screen "1.4.2_DR3_Advanced_Scale_Parameters_2" 800x480, template "Template_1"
   TextField "OBJECT_33" at 0,0 size 595x34; Text '1.4.2 Erweiterte Waagenparameter 2 von 5 / 1.4.2 Advanced Scale Parameter 2 of 5 / 1.4.2 Tous les paramètres 2/5 / Setup 1/3'
   Button "Exit_to_service_1" at 670,390 size 80x80; TextOn 'Texte / text'; TextOff 'Texte / text'; PictureOff "Right"
      on Press: ActivateScreen("1.4.3_DR3_Advanced_Scale_Parameters_3", 0)
   Button "Exit_to_service_2" at 545,390 size 80x80; TextOn 'Texte / text'; TextOff 'Texte / text'; PictureOff "Left"
      on Press: ActivateScreen("1.4.1_DR3_Advanced_Scale_Parameters_1", 0)
   Group "Group" at 700,5 size 95x30; Text 'Service'; PictureList "Signal_grey_yellow"
   Button "Exit_to_service" at 45,390 size 80x80; TextOn 'Texte / text'; TextOff 'Texte / text'; PictureOff "Exit"
      on Release: ActivateScreen("1.0_Menu_setup", 0)
      on Press: SetTag("WP231PR_DB_s_CMD2_i_CMD_CODE", '2'); SetBit("WP231PR_DB_s_CMD2_bo_CMD_TRIGGER")
   Button "OBJECT_13" at 360,390 size 80x80; TextOn 'Texte / text'; TextOff 'Texte / text'; PictureOff "Save"
      on Press: SetTag("WP231PR_DB_s_CMD2_i_CMD_CODE", '4003'); SetBit("WP231PR_DB_s_CMD2_bo_CMD_TRIGGER")
   TextField "OBJECT_306" at 172,114 size 279x26; Text 'Einschaltnullsetzen / Initial Zeroing / RAZ initiale / Scale name'
   TextField "OBJECT_7" at 69,155 size 380x26; Text 'Einschaltnullsetzen bei tarierter Waage / Initial zeroing if scale is tared / RAZ initiale quand la balance est tarée / Weight Unit'
   SymbolicIOField "Symbolisches EA-Feld_1" at 464,110 size 110x31; TextOn '1'; HelpText 'Die Waage kann durch einen Neustart automatisch nullgestellt werden. / The scale can be zeroed automatically by a power on. / La balance peut être remise à zéro à la mise sous tension'; TextOff '0'; TextList "003072_NO_YES"
      ProcessValue <- "WP231PR_DB_DR03_INITIAL_ZEROING"
   SymbolicIOField "Symbolisches EA-Feld_2" at 464,151 size 110x31; TextOn '1'; HelpText 'Shall the scale be zeroed by power on if it was tared? / RAZ à la mise sous tension lorsque la tare >< 0?'; TextOff '0'; TextList "003072_NO_YES"
      ProcessValue <- "WP231PR_DB_DR03_INITIAL_ZEROING_IF_TARED"
   TextField "OBJECT_3" at 25,199 size 426x26; Text 'Negativer Nullsetzgrenzwert (Einschaltnullsetzen) / Negative zeroing limit (initital zeroing) / Limite négative de RAZ (RAZ initiale) / Weight Unit'
      Visibility <- "WP231PR_DB_DR03_INITIAL_ZEROING"
   TextField "OBJECT_6" at 52,242 size 399x26; Text 'Positiver Nullsetzgrenzwert (Einschaltnullsetzen) / Positive zeroing limit (initial zeroing) / Limite positive de RAZ (RAZ initiale) / Weight Unit'
      Visibility <- "WP231PR_DB_DR03_INITIAL_ZEROING"
   IOField "OBJECT_28" at 464,191 size 110x40; HelpText 'Negative Begrenzung des Nullstellwerts nach Einschalten der Waage. / Limite négative de la RAZ à la mise sous tension'; FormatPattern 99.99
      ProcessValue <- "WP231PR_DB_DR03_INITIAL_ZEROING_LIM_NEG"
      Visibility <- "WP231PR_DB_DR03_INITIAL_ZEROING"
   IOField "OBJECT_8" at 464,235 size 110x40; HelpText 'Positive Begrenzung des Nullstellwerts nach Einschalten der Waage. / Plage RAZ positive après mise sous tension'; FormatPattern 99.99
      ProcessValue <- "WP231PR_DB_DR03_INITIAL_ZEROING_LIM_POS"
      Visibility <- "WP231PR_DB_DR03_INITIAL_ZEROING"
   TextField "OBJECT_2" at 194,75 size 257x26; Text 'Automatische Nullnachführung / Automatic Zero Tracking / Maintien du zéro (zéro suiveur) / Weight Unit'
   SymbolicIOField "Symbolisches EA-Feld_3" at 464,71 size 110x31; TextOn '1'; HelpText 'Driftet die Waage weniger als 1/4d pro Sekunde stellt sie automatisch null. ACHTUNG: Bei langsamer Drift kann eine volle Waage mit 0kg angezeigt werden! If the scale drifts less than 1/4d per second, it'll be zeroed automatically. ATTENTION: A slow drift can effect, that the scale shows 0kg even if it's full! La balance effectue automatiquement une RAZ quand le poids dérive de moins de 1/4d par sec'; TextOff '0'; TextList "003072_NO_YES"
      ProcessValue <- "WP231PR_DB_DR03_ZERO_TRACKING"
   TextField "OBJECT_4" at 12,330 size 440x26; Text 'Positiver Nullstellgrenzwert (halbselbstt. Nullstellen) / Positive zeroing limit (semi-automatic zeroing) / Limite positive de RAZ (RAZ semi-automatique) / Scale name'
   TextField "OBJECT_9" at 13,287 size 439x26; Text 'Negativer Nullstellgrenzwert (halbselbstt. Nullstellen) / Negative zeroing limit (semi-automatic zeroing) / Limite négative de RAZ (RAZ semi-automatique) / Weight Unit'
   IOField "OBJECT_10" at 464,323 size 110x40; HelpText 'Positive Begrenzung des Nullstellwerts der Waage. / Plage RAZ positive'; FormatPattern 99.99
      ProcessValue <- "WP231PR_DB_DR03_SEM_AUT_ZERO_LIM_POS"
   IOField "OBJECT_11" at 464,279 size 110x40; HelpText 'Negative Begrenzung des Nullstellwerts der Waage. / Limite négative de la RAZ'; FormatPattern 99.99
      ProcessValue <- "WP231PR_DB_DR03_SEM_AUT_ZERO_LIM_NEG"
   TextField "OBJECT_22" at 575,199 size 22x26; Text '% / Calibration Weight'
      Visibility <- "WP231PR_DB_DR03_INITIAL_ZEROING"
   TextField "OBJECT_1" at 576,243 size 22x26; Text '% / Calibration Weight'
      Visibility <- "WP231PR_DB_DR03_INITIAL_ZEROING"
   TextField "OBJECT_5" at 578,286 size 22x26; Text '% / Calibration Weight'
   TextField "OBJECT_12" at 577,331 size 22x26; Text '% / Calibration Weight'
   Group "Group_3" at 599,286 size 166x26; Text 'von'
   Group "Group_4" at 599,329 size 166x26; Text 'von'
   IOField "OBJECT_15" at 631,245 size 85x23; FormatPattern 9999999.9
      Visibility <- "WP231PR_DB_DR03_INITIAL_ZEROING"
      ProcessValue <- "WP231PR_DB_DR03_MAX_WEIGHT"
   TextField "Textfeld_2" at 599,243 size 30x25; Text 'von / of / de'
      Visibility <- "WP231PR_DB_DR03_INITIAL_ZEROING"
   IOField "I/O field_1" at 699,244 size 66x25; FormatPattern ????
      Visibility <- "WP231PR_DB_DR03_INITIAL_ZEROING"
      ProcessValue <- "WP231PR_DB_DR03_WEIGHT_UNIT"
   IOField "OBJECT_14" at 631,202 size 85x23; FormatPattern 9999999.9
      Visibility <- "WP231PR_DB_DR03_INITIAL_ZEROING"
      ProcessValue <- "WP231PR_DB_DR03_MAX_WEIGHT"
   TextField "Textfeld_1" at 599,200 size 30x25; Text 'von / of / de'
      Visibility <- "WP231PR_DB_DR03_INITIAL_ZEROING"
   IOField "I/O field_2" at 699,201 size 66x25; FormatPattern ????
      Visibility <- "WP231PR_DB_DR03_INITIAL_ZEROING"
      ProcessValue <- "WP231PR_DB_DR03_WEIGHT_UNIT"
   Softkey "[!Invalid!]Softkey_F6" at -140,-147 size 0x0
      on KeyDown: ActivateScreen("Menu_weighing_expert", 0)
   Softkey "[!Invalid!]Softkey_F5" at -140,-147 size 0x0
      on KeyDown: ActivateScreen("1.4.3_DR3_Advanced_Scale_Parameters_3", 0)
   GraphicIOField "OBJECT_19" at 765,5 size 30x30; PictureList "Signal_grey_yellow"
      ProcessValue <- "WP231PR_DB_s_IO_DATA_SCALE_STATUS_2_SERVICE_MODE"
   TextField "OBJECT_37" at 700,7 size 57x25; Text 'Service / Error occurred'
   IOField "OBJECT_16" at 631,288 size 85x23; FormatPattern 9999999.9
      ProcessValue <- "WP231PR_DB_DR03_MAX_WEIGHT"
   TextField "Textfeld_3" at 599,286 size 30x25; Text 'von / of / de'
   IOField "I/O field_3" at 699,287 size 66x25; FormatPattern ????
      ProcessValue <- "WP231PR_DB_DR03_WEIGHT_UNIT"
   IOField "OBJECT_17" at 631,331 size 85x23; FormatPattern 9999999.9
      ProcessValue <- "WP231PR_DB_DR03_MAX_WEIGHT"
   TextField "Textfeld_4" at 599,329 size 30x25; Text 'von / of / de'
   IOField "I/O field_4" at 699,330 size 66x25; FormatPattern ????
      ProcessValue <- "WP231PR_DB_DR03_WEIGHT_UNIT"

screen "1.4.3_DR3_Advanced_Scale_Parameters_3" 800x480, template "Template_1"
   TextField "OBJECT_33" at 0,0 size 595x34; Text '1.4.3 Erweiterte Waagenparameter 3 von 5 / 1.4.3 Advanced Scale Parameter 3 of 5 / 1.4.3 Tous les paramètres 3/5 / Setup 1/3'
   TextField "OBJECT_306" at 111,200 size 122x26; Text 'Tarahöchstlast / Tare maximum / Tare max / Scale name'
   IOField "OBJECT_307" at 238,193 size 371x40; HelpText 'Limitation of the tare weight. / Limitation de la valeur de la tare'; FormatPattern 999.99
      ProcessValue <- "WP231PR_DB_DR03_TARE_MAX"
   TextField "OBJECT_6" at 2,143 size 234x26; Text 'Gewichtssimulation zulassen / Weight Simulation enabled / Autoriser simulation du poids / Scale name'
   TextField "OBJECT_11" at 6,70 size 227x26; Text 'Runden der Prozesswerte / Rounding for process values / Arrondi valeurs processus / Scale name'
   TextField "OBJECT_7" at 117,106 size 116x26; Text 'Additives Tara / Additive tare / Tare additive / Weight Unit'
   SymbolicIOField "Symbolisches EA-Feld_4" at 239,105 size 371x31; TextOn '1'; HelpText 'Works the scale with additive tare? / Utilisation de la tare additive?'; TextOff '0'; TextList "003072_NO_YES"
      ProcessValue <- "WP231PR_DB_DR03_ADDITIVE_TARE"
   SymbolicIOField "Symbolisches EA-Feld_5" at 239,140 size 371x33; TextOn '1'; HelpText 'Should the weight simulation be possible? / Simulation du poids autorisée?'; TextOff '0'; TextList "003072_NO_YES"
      ProcessValue <- "WP231PR_DB_DR03_WEIGHT_SIM_ALLOWED"
   SymbolicIOField "Symbolisches EA-Feld_6" at 239,67 size 371x33; TextOn '1'; HelpText 'Runding of the internal process values of the scale. These are independent from the resolution step of the scale. / Arrondi valeurs processus internes. Indépendant de la résolution de la balance'; TextOff '0'; TextList "003074_ROUNDING_PROCESS_VAL"
      ProcessValue <- "WP231PR_DB_DR03_DEC_POINT_PROC_VAL"
   TextField "OBJECT_2" at 96,245 size 140x26; Text 'Stillstandsbereich / Standstill range / Plage état stable / Scale name'
   TextField "OBJECT_3" at 93,291 size 145x26; Text 'Stillstandszeit / Standstill time / Temps état stable / Weight Unit'
   IOField "OBJECT_4" at 238,238 size 371x40; HelpText 'Stillstandswert in "d" (=Ziffernschritt) / Standstill range in "d" (=Resolution Step) / Plage état stable (d) d =résolution'; FormatPattern 999
      ProcessValue <- "WP231PR_DB_DR03_ST_STILL_RANGE_D"
   IOField "OBJECT_28" at 238,282 size 371x40; HelpText 'Standstill time in seconds / Temps état stable en secondes'; FormatPattern 999999
      ProcessValue <- "WP231PR_DB_DR03_ST_STILL_TIME"
   TextField "OBJECT_23" at 612,200 size 22x26; Text '% / Calibration Weight'
   TextField "OBJECT_1" at 613,289 size 12x26; Text 's / Calibration Weight'
   TextField "OBJECT_5" at 30,333 size 204x26; Text 'Stillstandswartezeit / Standstill delay time / Temporisation état stable / Weight Unit'
   TextField "OBJECT_8" at 613,332 size 12x26; Text 's / Calibration Weight'
   IOField "OBJECT_9" at 238,326 size 371x40; HelpText 'Standstill delay time in seconds / Temporisation état stable en secondes'; FormatPattern 999999
      ProcessValue <- "WP231PR_DB_DR03_ST_STILL_WAITING_TIME"
   Button "Exit_to_service_1" at 670,390 size 80x80; TextOn 'Texte / text'; TextOff 'Texte / text'; PictureOff "Right"
      on Press: ActivateScreen("1.4.4_DR3_Advanced_Scale_Parameters_4", 0)
   Button "Exit_to_service_2" at 545,390 size 80x80; TextOn 'Texte / text'; TextOff 'Texte / text'; PictureOff "Left"
      on Press: ActivateScreen("1.4.2_DR3_Advanced_Scale_Parameters_2", 0)
   Group "Group" at 700,5 size 95x30; Text 'Service'; PictureList "Signal_grey_yellow"
   Button "Exit_to_service" at 45,390 size 80x80; TextOn 'Texte / text'; TextOff 'Texte / text'; PictureOff "Exit"
      on Release: ActivateScreen("1.0_Menu_setup", 0)
      on Press: SetTag("WP231PR_DB_s_CMD2_i_CMD_CODE", '2'); SetBit("WP231PR_DB_s_CMD2_bo_CMD_TRIGGER")
   Button "OBJECT_10" at 360,390 size 80x80; TextOn 'Texte / text'; TextOff 'Texte / text'; PictureOff "Save"
      on Press: SetTag("WP231PR_DB_s_CMD2_i_CMD_CODE", '4003'); SetBit("WP231PR_DB_s_CMD2_bo_CMD_TRIGGER")
   TextField "OBJECT_12" at 611,244 size 14x26; Text 'd / Calibration Weight'
   IOField "OBJECT_14" at 666,203 size 85x23; FormatPattern 9999999.9
      ProcessValue <- "WP231PR_DB_DR03_MAX_WEIGHT"
   TextField "Textfeld_1" at 634,201 size 30x25; Text 'von / of / de'
   IOField "I/O field_2" at 734,202 size 66x25; FormatPattern ????
      ProcessValue <- "WP231PR_DB_DR03_WEIGHT_UNIT"
   Softkey "[!Invalid!]Softkey_F6" at -140,-147 size 0x0
      on KeyDown: ActivateScreen("Menu_weighing_expert", 0)
   Softkey "[!Invalid!]Softkey_F5" at -140,-147 size 0x0
      on KeyDown: ActivateScreen("1.4.4_DR3_Advanced_Scale_Parameters_4", 0)
   Softkey "[!Invalid!]Softkey_F4" at -140,-147 size 0x0
      on KeyDown: ActivateScreen("1.4.2_DR3_Advanced_Scale_Parameters_2", 0)
   GraphicIOField "OBJECT_19" at 765,5 size 30x30; PictureList "Signal_grey_yellow"
      ProcessValue <- "WP231PR_DB_s_IO_DATA_SCALE_STATUS_2_SERVICE_MODE"
   TextField "OBJECT_37" at 700,7 size 57x25; Text 'Service / Error occurred'

screen "1.4.4_DR3_Advanced_Scale_Parameters_4" 800x480, template "Template_1"
   TextField "OBJECT_33" at 0,0 size 595x34; Text '1.4.4 Erweiterte Waagenparameter 4 von 5 / 1.4.4 Advanced Scale Parameter 4 of 5 / 1.4.4 Tous les paramètres 4/5 / Setup 1/3'
   TextField "OBJECT_6" at 141,103 size 304x32; Text 'Grenzfrequenz Tiefpassfilter 1 / Frequency low pass filter 1 / Filtre passe-bas 1 / Weight Unit'
   IOField "OBJECT_8" at 457,99 size 110x40; HelpText 'Frequenz Tiefpassfilter 1. Bei hohen Frequenzen reagiert die Waage sehr schnell, bei niedrigen träger. / Frequency of low pass filter 1. A high frequency makes the scale fast, a small more sluggish. / Filtre passe bas 1. Une valeur élevée rend la balance plus réactive'; FormatPattern 99.9
      ProcessValue <- "WP231PR_DB_DR03_FREQ_LOW_PASS_1"
   IOField "OBJECT_5" at 456,238 size 110x40; HelpText 'Frequenz Tiefpassfilter 2. Bei hohen Frequenzen reagiert die Waage sehr schnell, bei niedrigen träger. / Filtre passe bas 2. Une valeur élevée rend la balance plus réactive'; FormatPattern 99.9
      ProcessValue <- "WP231PR_DB_DR03_FREQ_LOW_PASS_2"
   TextField "OBJECT_4" at 149,149 size 297x32; Text 'Ordnungszahl Tiefpassfilter 1 / Order no low pass filter 1 / Ordre filtre passe-bas 1 / Weight Unit'
   TextField "OBJECT_9" at 149,288 size 297x32; Text 'Ordnungszahl Tiefpassfilter 2 / Order no low pass filter 2 / Ordre filtre passe-bas 2 / Weight Unit'
   TextField "OBJECT_12" at 164,195 size 283x32; Text 'Tiefe Mittelwertfilter / Depth of the average filter / Filtre des valeurs moyennes / Weight Unit'
   IOField "OBJECT_13" at 456,189 size 110x40; HelpText 'Die Waage errechnet intern alle 10ms einen neuen Gewichtswert. Der Mittelwert filter bildet dann über X Werte einen fortlaufenden Mittelwert. / The scale creates internally each 10ms a new weight value. The average filter then creates an continuous average of X values. / La balance calcule une valeur moyenne glissante sur "X" valeurs'; FormatPattern 999
      ProcessValue <- "WP231PR_DB_DR03_AVER_FILTER_DEPTH"
   SymbolicIOField "Symbolisches EA-Feld_1" at 457,148 size 110x34; TextOn '1'; HelpText 'Ordnungszahl Tiefpassfilter 1. / Ordre filtre passe-bas 1'; TextOff '0'; TextList "003112_ORDER_NO_LOW_PASS_FILTER"
      ProcessValue <- "WP231PR_DB_DR03_ORDER_NO_LOW_PASS_1"
   SymbolicIOField "Symbolisches EA-Feld_2" at 456,288 size 110x34; TextOn '1'; HelpText 'Ordnungszahl Tiefpassfilter 2. / Ordre filtre passe-bas 2'; TextOff '0'; TextList "003112_ORDER_NO_LOW_PASS_FILTER"
      ProcessValue <- "WP231PR_DB_DR03_ORDER_NO_LOW_PASS_2"
   TextField "OBJECT_3" at 144,240 size 304x32; Text 'Grenzfrequenz Tiefpassfilter 2 / Frequency low pass filter 2 / Filtre passe-bas 2 / Weight Unit'
   Button "OBJECT_1" at 360,390 size 80x80; TextOn 'Texte / text'; TextOff 'Texte / text'; PictureOff "Save"
      on Press: SetTag("WP231PR_DB_s_CMD2_i_CMD_CODE", '4003'); SetBit("WP231PR_DB_s_CMD2_bo_CMD_TRIGGER")
   Button "Exit_to_service_2" at 545,390 size 80x80; TextOn 'Texte / text'; TextOff 'Texte / text'; PictureOff "Left"
      on Press: ActivateScreen("1.4.3_DR3_Advanced_Scale_Parameters_3", 0)
   Group "Group" at 700,5 size 95x30; Text 'Service'; PictureList "Signal_grey_yellow"
   Button "Exit_to_service" at 45,390 size 80x80; TextOn 'Texte / text'; TextOff 'Texte / text'; PictureOff "Exit"
      on Release: ActivateScreen("1.0_Menu_setup", 0)
      on Press: SetTag("WP231PR_DB_s_CMD2_i_CMD_CODE", '2'); SetBit("WP231PR_DB_s_CMD2_bo_CMD_TRIGGER")
   TextField "Textfeld_1" at 572,107 size 23x25; Text 'Hz'
   TextField "Textfeld_2" at 572,247 size 23x25; Text 'Hz'
   Softkey "[!Invalid!]Softkey_F6" at -140,-147 size 0x0
      on KeyDown: ActivateScreen("Menu_weighing_expert", 0)
   Softkey "[!Invalid!]Softkey_F5" at -140,-147 size 0x0
      on KeyDown: SetTag("S1_CMD2.i_CMD_CODE", 4003); SetTag("S1_CMD2.i_CMD_TRIGGER", 1)
   Softkey "[!Invalid!]Softkey_F4" at -140,-147 size 0x0
      on KeyDown: ActivateScreen("1.4.3_DR3_Advanced_Scale_Parameters_3", 0)
   GraphicIOField "OBJECT_19" at 765,5 size 30x30; PictureList "Signal_grey_yellow"
      ProcessValue <- "WP231PR_DB_s_IO_DATA_SCALE_STATUS_2_SERVICE_MODE"
   TextField "OBJECT_37" at 700,7 size 57x25; Text 'Service / Error occurred'

screen "2.2.2_Scale_Status_2_DR5" 800x480, template "Template_1"
   TextField "OBJECT_33" at 0,0 size 387x34; Text '2.2.2 Waagenstatus 2 von 4 / 2.2.2 Scale Status 2 of 4 / 2.2.2 Etat de la balance 2/4 / Setup 1/3'
   TextField "OBJECT_306" at 117,91 size 387x26; Text 'Tara (Vorgabe) / Current tare weight (preset tare) / Valeur actuelle tare (prédétermination de la tare) / Scale name'
   IOField "OBJECT_307" at 515,84 size 195x40; FormatPattern 999999.9999
      ProcessValue <- "WP231PR_DB_DR05_TARE_WEIGHT_PRESET"
   TextField "OBJECT_7" at 189,142 size 315x26; Text 'Tara (halbselbsttätig) / Current tare weight (semi-automatic) / Valeur actuelle tare (semi-automatique) / Weight Unit'
   IOField "OBJECT_28" at 515,134 size 195x40; FormatPattern 999999.9999
      ProcessValue <- "WP231PR_DB_DR05_TARE_WEIGHT_SEM_AUT"
   Button "OBJECT_24" at 45,390 size 80x80; TextOn 'Texte / text'; TextOff 'Texte / text'; PictureOff "Exit"
      on Press: ActivateScreen("2.0_Menu_diagnostic", 0); SetTag("WP231PR_DB_CMD_B", 0)
   TextField "OBJECT_6" at 197,192 size 307x26; Text 'Einschaltnullsetzwert / Current zeroing weight (initial zeroing) / Valeur actuelle du zéro (RAZ initiale) / Weight Unit'
   IOField "OBJECT_8" at 515,185 size 195x40; FormatPattern 999999.9999
      ProcessValue <- "WP231PR_DB_DR05_ZEROING_WEIGHT_INITIAL"
   TextField "OBJECT_2" at 198,295 size 304x26; Text 'Nullstellwert (Nullnachführung) / Current zeroing weight (zero tracking) / Valeur actuelle du zéro (zéro suiveur) / Scale name'
   IOField "OBJECT_5" at 515,289 size 195x40; FormatPattern 999999.9999
      ProcessValue <- "WP231PR_DB_DR05_ZEROING_WEIGHT_TRACKING"
   IOField "OBJECT_9" at 515,340 size 195x40; FormatPattern 999999.9999
      ProcessValue <- "WP231PR_DB_DR05_DEAD_LOAD"
   TextField "OBJECT_11" at 320,345 size 185x26; Text 'Totlast (errechnet) / Dead Load (calculated) / Poids mort (calculé) / Scale name'
   TextField "OBJECT_4" at 122,244 size 382x26; Text 'Nullstellwert (halbselbsttätig) / Current zeroing weight (semi-automatic) / Valeur actuelle du zéro (RAZ semi-automatique) / Weight Unit'
   IOField "OBJECT_10" at 515,237 size 195x40; FormatPattern 999999.9999
      ProcessValue <- "WP231PR_DB_DR05_ZEROING_WEIGHT_SEM_AUT"
   IOField "I/O field_2" at 710,92 size 74x25; FormatPattern ????
      ProcessValue <- "WP231PR_DB_DR03_WEIGHT_UNIT"
   IOField "I/O field_1" at 710,142 size 74x25; FormatPattern ????
      ProcessValue <- "WP231PR_DB_DR03_WEIGHT_UNIT"
   IOField "I/O field_3" at 710,192 size 74x25; FormatPattern ????
      ProcessValue <- "WP231PR_DB_DR03_WEIGHT_UNIT"
   IOField "I/O field_4" at 710,245 size 74x25; FormatPattern ????
      ProcessValue <- "WP231PR_DB_DR03_WEIGHT_UNIT"
   IOField "I/O field_5" at 710,298 size 74x25; FormatPattern ????
      ProcessValue <- "WP231PR_DB_DR03_WEIGHT_UNIT"
   IOField "I/O field_6" at 710,348 size 74x25; FormatPattern ????
      ProcessValue <- "WP231PR_DB_DR03_WEIGHT_UNIT"
   IOField "OBJECT_301" at 0,40 size 800x40; FormatPattern ????????????????
      ProcessValue <- "WP231PR_DB_DR34_ASCII_DISPLAY"
   Button "OBJECT_1" at 670,390 size 80x80; TextOn 'Texte / text'; TextOff 'Texte / text'; PictureOff "Right"
      on Press: ActivateScreen("2.2.3_Scale_Status_3_DR30", 0); SetTag("WP231PR_DB_CMD_B", 2030)
   Button "OBJECT_25" at 545,390 size 80x80; TextOn 'Texte / text'; TextOff 'Texte / text'; PictureOff "Left"
      on Press: ActivateScreen("2.2.1_Scale_Status_1", 0)
   Button "Up_to Setup_5_Min_2" at 360,390 size 80x80; TextOn 'Texte / text'; TextOff 'Texte / text'; PictureOff "Home_3"
      on Press: ActivateScreen("0.0.0_Scale_View_1", 0); SetTag("WP231PR_DB_CMD_B", 0)
   Softkey "[!Invalid!]Softkey_F6" at -140,-147 size 0x0
      on KeyDown: ActivateScreen("2.0_Menu_diagnostic", 0)

screen "1.5.1.1_DR7_digital_in_outputs_1" 800x480, template "Template_1"
   TextField "OBJECT_33" at 0,0 size 766x34; Text '1.5.1.1 Einstellungen Digital Ein- und Ausgänge 1 von 2 / 1.5.1.1 Digital In- and Outputs Settings 1 of 2 / 1.5.1.1 Paramétrage E/S TOR 1/2 / Setup 1/3'
   TextField "OBJECT_306" at 20,96 size 154x34; Text 'Eingang DI.0 / Input DI.0 / Entrée TOR 0 / Scale name'
   Button "OBJECT_34" at 670,390 size 80x80; TextOn 'Texte / text'; TextOff 'Texte / text'; PictureOff "Right"
      on Release: ActivateScreen("1.5.1.2_DR7_digital_in_outputs_2", 0)
   Button "OBJECT_24" at 45,390 size 80x80; TextOn 'Texte / text'; TextOff 'Texte / text'; PictureOff "Exit"
      on Release: ActivateScreen("1.5.0.1_Menu_communication_interfaces_1", 0)
   TextField "OBJECT_6" at 20,219 size 154x34; Text 'Eingang DI.2 / Input DI.2 / Entrée TOR 2 / Weight Unit'
   TextField "OBJECT_2" at 20,336 size 264x34; Text 'Filterung der Eingänge / Filter digital input / Filtre pour entrées TOR / Scale name'
   TextField "OBJECT_4" at 20,277 size 154x34; Text 'Eingang DI.3 / Input DI.3 / Entrée TOR 3 / Weight Unit'
   TextField "OBJECT_7" at 20,159 size 154x34; Text 'Eingang DI.1 / Input DI.1 / Entrée TOR 1 / Scale name'
   TextField "OBJECT_9" at 321,56 size 319x30; Text 'Funktionszuweisung / Functions for Digital Inputs / Affectation de la fonction / Scale name'
   SymbolicIOField "Symbolisches EA-Feld_1" at 289,96 size 390x36; TextOn '1'; TextOff '0'; TextList "007008_ASSIGNMENT_DIGITAL_INPUT"
      ProcessValue <- "WP231PR_DB_DR07_ASSIGN_DI_0"
   SymbolicIOField "Symbolisches EA-Feld_2" at 289,159 size 390x36; TextOn '1'; TextOff '0'; TextList "007008_ASSIGNMENT_DIGITAL_INPUT"
      ProcessValue <- "WP231PR_DB_DR07_ASSIGN_DI_1"
   SymbolicIOField "Symbolisches EA-Feld_3" at 289,219 size 390x36; TextOn '1'; TextOff '0'; TextList "007008_ASSIGNMENT_DIGITAL_INPUT"
      ProcessValue <- "WP231PR_DB_DR07_ASSIGN_DI_2"
   SymbolicIOField "Symbolisches EA-Feld_4" at 289,277 size 390x36; TextOn '1'; TextOff '0'; TextList "007008_ASSIGNMENT_DIGITAL_INPUT"
      ProcessValue <- "WP231PR_DB_DR07_ASSIGN_DI_3"
   SymbolicIOField "Symbolisches EA-Feld_5" at 289,336 size 390x36; TextOn '1'; TextOff '0'; TextList "007016_FILTER_DIGITAL_INPUT"
      ProcessValue <- "WP231PR_DB_DR07_FILTER_DI"
   Button "OBJECT_3" at 420,390 size 80x80; TextOn 'Texte / text'; TextOff 'Texte / text'; PictureOff "Save"
      on Press: SetTag("WP231PR_DB_s_CMD2_i_CMD_CODE", '4007'); SetBit("WP231PR_DB_s_CMD2_bo_CMD_TRIGGER")
   Softkey "[!Invalid!]Softkey_F6" at -140,-147 size 0x0
      on KeyDown: ActivateScreen("1.5.0.1_Menu_communication_interfaces_1", 0)
   Softkey "[!Invalid!]Softkey_F5" at -140,-147 size 0x0
      on KeyDown: ActivateScreen("1.5.1.2_DR7_digital_in_outputs_2", 0)

screen "1.5.2_DR7_Analogue_Output" 800x480, template "Template_1"
   TextField "OBJECT_33" at 0,0 size 464x34; Text '1.5.2 Einstellungen Analogausgang / 1.5.2 Analogue Output Settings / 1.5.2 Paramétrage sortie analogique / Setup 1/3'
   Button "OBJECT_24" at 45,390 size 80x80; TextOn 'Texte / text'; TextOff 'Texte / text'; PictureOff "Exit"
      on Release: ActivateScreen("1.5.0.1_Menu_communication_interfaces_1", 0)
   Button "OBJECT_6" at 360,390 size 80x80; TextOn 'Texte / text'; TextOff 'Texte / text'; PictureOff "Save"
      on Press: SetTag("WP231PR_DB_s_CMD2_i_CMD_CODE", '4007'); SetBit("WP231PR_DB_s_CMD2_bo_CMD_TRIGGER")
   TextField "OBJECT_4" at 12,320 size 339x32; Text 'Ersatzwert bei Störung oder Stop / Defined value by error or stop / Valeur remplacement si erreur / Weight Unit'
      Visibility <- "WP231PR_DB_DR07_ANA_OUT_BY_ERR_OR_STOP_1"
   IOField "OBJECT_5" at 360,316 size 315x40; FormatPattern 99.99
      ProcessValue <- "WP231PR_DB_DR07_ANA_OUT_ERR"
      Visibility <- "WP231PR_DB_DR07_ANA_OUT_BY_ERR_OR_STOP_1"
   TextField "OBJECT_1" at 687,325 size 44x32; Text 'mA / Weight Unit'
      Visibility <- "WP231PR_DB_DR07_ANA_OUT_BY_ERR_OR_STOP_1"
   TextField "OBJECT_11" at 270,82 size 79x32; Text 'Bereich / Range / Plage / Scale name'
   TextField "OBJECT_12" at 90,273 size 262x32; Text 'Störungs-/Stop-Verhalten / Status by error or stop / Erreur - Stop / Weight Unit'
   TextField "OBJECT_13" at 90,177 size 266x32; Text 'Startwert (0/4mA) / Start value / Valeur de départ (0/4mA) / Weight Unit'
   TextField "OBJECT_14" at 275,129 size 73x32; Text 'Quelle / Source / Scale name'
   IOField "OBJECT_18" at 361,173 size 315x40; FormatPattern 999999.999
      ProcessValue <- "WP231PR_DB_DR07_START_VAL_ANA_OUT"
   TextField "OBJECT_2" at 141,226 size 216x32; Text 'Endwert (20mA) / End value / Valeur de fin (20mA) / Weight Unit'
   IOField "OBJECT_3" at 360,222 size 315x40; FormatPattern 999999.999
      ProcessValue <- "WP231PR_DB_DR07_END_VAL_ANA_OUT"
   SymbolicIOField "Symbolisches EA-Feld_1" at 362,126 size 347x34; TextOn '1'; TextOff '0'; TextList "007032_SOURCE_ANALOG_OUTPUT"
      ProcessValue <- "WP231PR_DB_DR07_SOURCE_ANA_OUT"
   SymbolicIOField "Symbolisches EA-Feld_2" at 360,271 size 382x34; TextOn '1'; TextOff '0'; TextList "007034_ANALOG_STATUS_BY_ERROR_STOP"
      ProcessValue <- "WP231PR_DB_DR07_ANA_OUT_BY_ERR_OR_STOP_1"
   SymbolicIOField "Symbolisches EA-Feld_3" at 362,80 size 382x34; TextOn '1'; TextOff '0'; TextList "007030_RANGE_ANALOG_OUTPUT"
      ProcessValue <- "WP231PR_DB_DR07_RANGE_ANA_OUT"
   IOField "I/O field_2" at 682,174 size 60x40; FormatPattern ????
      ProcessValue <- "WP231PR_DB_DR03_WEIGHT_UNIT"
   IOField "I/O field_1" at 682,222 size 60x40; FormatPattern ????
      ProcessValue <- "WP231PR_DB_DR03_WEIGHT_UNIT"
   Softkey "[!Invalid!]Softkey_F6" at -140,-147 size 0x0
      on KeyDown: ActivateScreen("1.5.0.1_Menu_communication_interfaces_1", 0)
   Softkey "[!Invalid!]Softkey_F5" at -140,-147 size 0x0
      on KeyDown: ActivateScreen("1.5.7_DR7_trace_settings", 0)
   Softkey "[!Invalid!]Softkey_F4" at -140,-147 size 0x0
      on KeyDown: ActivateScreen("DR7_Process_Interfaces_3", 0)

screen "1.5.7_DR7_trace_settings" 800x480, template "Template_1"
   TextField "OBJECT_33" at 0,0 size 348x34; Text '1.5.7 Trace Einstellungen / 1.5.7 Trace Settings / 1.5.7 Paramètres Trace / Setup 1/3'
   Button "OBJECT_34" at 360,390 size 80x80; TextOn 'Texte / text'; TextOff 'Texte / text'; PictureOff "Save"
      on Press: SetTag("WP231PR_DB_s_CMD2_i_CMD_CODE", '4007'); SetBit("WP231PR_DB_s_CMD2_bo_CMD_TRIGGER")
   Button "OBJECT_24" at 45,390 size 80x80; TextOn 'Texte / text'; TextOff 'Texte / text'; PictureOff "Exit"
      on Press: ActivateScreen("1.5.0.2_Menu_communication_interfaces_2", 0)
   Button "Schaltfläche_1" at 110,286 size 580x70; TextOn 'Texte'; TextOff 'Lösche Trace Speicher / Delete Trace Mememory / Effacer la mémoire trace'
      on Press: SetTag("WP231PR_DB_s_CMD2_i_CMD_CODE", '454'); SetBit("WP231PR_DB_s_CMD2_bo_CMD_TRIGGER")
   TextField "OBJECT_11" at 110,121 size 211x32; Text 'Aufzeichnungszyklus / Trace rate / Durée cycle trace / Scale name'
   SymbolicIOField "Symbolisches EA-Feld_1" at 328,122 size 430x34; TextOn '1'; TextOff '0'; TextList "007048_TRACE_RATE"
      ProcessValue <- "WP231PR_DB_DR07_TRACE_RATE"
   TextField "OBJECT_13" at 111,204 size 186x32; Text 'Speichermethode / Memory type / Méthode mémoire / Weight Unit'
   SymbolicIOField "Symbolisches EA-Feld_2" at 328,204 size 430x34; TextOn '1'; TextOff '0'; TextList "007050_TRACE_MEMORY_TYPE"
      ProcessValue <- "WP231PR_DB_DR07_TRACE_MEM_TYPE"
   Button "Up_to Setup_5_Min_2" at 678,390 size 80x80; TextOn 'Texte / text'; TextOff 'Texte / text'; PictureOff "Home_3"
      on Release: ActivateScreen("0.0.0_Scale_View_1", 0)
   Softkey "[!Invalid!]Softkey_F6" at -140,-147 size 0x0
      on KeyDown: ActivateScreen("1.5.0.1_Menu_communication_interfaces_1", 0)
   Softkey "[!Invalid!]Softkey_F5" at -140,-147 size 0x0
      on KeyDown: SetTag("S1_CMD2.i_CMD_CODE", 4007); SetTag("S1_CMD2.i_CMD_TRIGGER", 1)
   Softkey "[!Invalid!]Softkey_F4" at -140,-147 size 0x0
      on KeyDown: ActivateScreen("1.5.2_DR7_Analogue_Output", 0)

screen "1.5.8_DR12_Ethernet_parameters" 800x480, template "Template_1"
   TextField "OBJECT_33" at 0,0 size 379x34; Text '1.5.8 Ethernet Parameter / 1.5.8 Ethernet Settings / 1.5.8 Paramétrage Ethernet / Setup 1/3'
   TextField "OBJECT_306" at 69,111 size 135x32; Text 'Mac Adresse / MAC address / Adresse Mac / Scale name'
   IOField "OBJECT_307" at 125,150 size 100x50; FormatPattern FFFF
      ProcessValue <- "WP231PR_DB_DR12_DEVICE_MAC_ADDRESS"
   Button "OBJECT_24" at 45,390 size 80x80; TextOn 'Texte / text'; TextOff 'Texte / text'; PictureOff "Exit"
      on Release: SetTag("WP231PR_DB_s_CMD2_i_CMD_CODE", 2); SetBit("WP231PR_DB_s_CMD2_bo_CMD_TRIGGER")
      on Press: ActivateScreen("1.5.0.2_Menu_communication_interfaces_2", 0)
   TextField "OBJECT_6" at 70,246 size 112x32; Text 'IP Adresse / IP address / Adresse IP / Weight Unit'
   IOField "OBJECT_8" at 125,282 size 100x50; FormatPattern 999
      ProcessValue <- "WP231PR_DB_DR12_IP_ADDRESS_1"
   IOField "OBJECT_3" at 228,150 size 100x50; FormatPattern FFFF
      ProcessValue <- "WP231PR_DB_DR12_DEVICE_MAC_ADDRESS_1"
   IOField "OBJECT_4" at 330,150 size 100x50; FormatPattern FFFF
      ProcessValue <- "WP231PR_DB_DR12_DEVICE_MAC_ADDRESS_2"
   IOField "OBJECT_5" at 432,150 size 100x50; FormatPattern FFFF
      ProcessValue <- "WP231PR_DB_DR12_DEVICE_MAC_ADDRESS_3"
   IOField "OBJECT_9" at 535,150 size 100x50; FormatPattern FFFF
      ProcessValue <- "WP231PR_DB_DR12_DEVICE_MAC_ADDRESS_4"
   IOField "OBJECT_10" at 638,150 size 100x50; FormatPattern FFFF
      ProcessValue <- "WP231PR_DB_DR12_DEVICE_MAC_ADDRESS_5"
   IOField "OBJECT_17" at 228,282 size 100x50; FormatPattern 999
      ProcessValue <- "WP231PR_DB_DR12_IP_ADDRESS_2"
   IOField "OBJECT_18" at 330,282 size 100x50; FormatPattern 999
      ProcessValue <- "WP231PR_DB_DR12_IP_ADDRESS_3"
   IOField "OBJECT_19" at 432,282 size 100x50; FormatPattern 999
      ProcessValue <- "WP231PR_DB_DR12_IP_ADDRESS_4"
   Button "Up_to Setup_5_Min_2" at 658,390 size 80x80; TextOn 'Texte / text'; TextOff 'Texte / text'; PictureOff "Home_3"
      on Release: ActivateScreen("0.0.0_Scale_View_1", 0)
      on Press: SetTag("WP231PR_DB_s_CMD2_i_CMD_CODE", 2); SetBit("WP231PR_DB_s_CMD2_bo_CMD_TRIGGER")
   Button "OBJECT_1" at 360,390 size 80x80; TextOn 'Texte / text'; TextOff 'Texte / text'; PictureOff "Save"
      on Release: SetTag("WP231PR_DB_s_CMD2_i_CMD_CODE", '4012'); SetBit("WP231PR_DB_s_CMD2_bo_CMD_TRIGGER")
   Softkey "[!Invalid!]Softkey_F6" at -140,-147 size 0x0
      on KeyDown: ActivateScreen("Menu_interfaces", 0)

screen "1.5.6_DR13_RS485-Parameter" 800x480, template "Template_1"
   TextField "OBJECT_33" at 0,0 size 339x34; Text '1.5.6 RS485 Parameter / 1.5.6 RS485 Settings / 1.5.6 Paramètres RS485 / Setup 1/3'
   TextField "OBJECT_306" at 260,81 size 84x29; Text 'Protokoll / Protocol / Rapport / Scale name'
   TextField "OBJECT_7" at 125,125 size 222x29; Text 'Baudrate / Baud rate / Vitesse de transmission / Weight Unit'
      Visibility <- "WP231PR_DB_DR13_RS485_PROTOCOL"
   Button "OBJECT_24" at 45,390 size 80x80; TextOn 'Texte / text'; TextOff 'Texte / text'; PictureOff "Exit"
      on Press: ActivateScreen("1.5.0.1_Menu_communication_interfaces_1", 0)
   TextField "OBJECT_6" at 205,169 size 138x29; Text 'Zeichenparität / Parity / Parité / Weight Unit'
      Visibility <- "WP231PR_DB_DR13_RS485_PROTOCOL"
   TextField "OBJECT_2" at 182,212 size 161x29; Text 'Anzahl Datenbits / Data bits / Bits de données / Scale name'
      Visibility <- "WP231PR_DB_DR13_RS485_PROTOCOL"
   TextField "OBJECT_4" at 143,295 size 202x29; Text 'Modbusadresse RTU / Modbus address RTU / Adresse Modbus RTU / Weight Unit'
      Visibility <- "WP231PR_DB_DR13_RS485_PROTOCOL"
   IOField "OBJECT_10" at 350,295 size 320x30; FormatPattern 99999
      ProcessValue <- "WP231PR_DB_DR13_MODBUS_RTU_ADDRESS"
      Visibility <- "WP231PR_DB_DR13_RS485_PROTOCOL"
   TextField "OBJECT_11" at 25,335 size 322x29; Text 'Kommastelle Fernanzeige / Decimal point remote display / Point décimal afficheur à distance / Weight Unit'
      Visibility <- "WP231PR_DB_DR13_RS485_PROTOCOL"
   Button "OBJECT_1" at 360,390 size 80x80; TextOn 'Texte / text'; TextOff 'Texte / text'; PictureOff "Save"
      on Release: SetTag("WP231PR_DB_s_CMD2_i_CMD_CODE", '4013'); SetBit("WP231PR_DB_s_CMD2_bo_CMD_TRIGGER")
   SymbolicIOField "Symbolisches EA-Feld_1" at 350,80 size 320x31; TextOn '1'; TextOff '0'; TextList "013008_RS485_PROTOCOL"
      ProcessValue <- "WP231PR_DB_DR13_RS485_PROTOCOL"
   SymbolicIOField "Symbolisches EA-Feld_2" at 350,125 size 320x31; TextOn '1'; TextOff '0'; TextList "013010_RS485_BAUD_RATE"
      ProcessValue <- "WP231PR_DB_DR13_RS485_BAUD_RATE"
      Visibility <- "WP231PR_DB_DR13_RS485_PROTOCOL"
   SymbolicIOField "Symbolisches EA-Feld_3" at 350,169 size 320x31; TextOn '1'; TextOff '0'; TextList "013012_RS485_PARITY"
      ProcessValue <- "WP231PR_DB_DR13_RS485_PARITY"
      Visibility <- "WP231PR_DB_DR13_RS485_PROTOCOL"
   SymbolicIOField "Symbolisches EA-Feld_4" at 350,212 size 320x31; TextOn '1'; TextOff '0'; TextList "013012_RS485_DATA_BITS"
      ProcessValue <- "WP231PR_DB_DR13_RS485_DATA_BITS"
      Visibility <- "WP231PR_DB_DR13_RS485_PROTOCOL"
   SymbolicIOField "Symbolisches EA-Feld_5" at 350,335 size 320x31; TextOn '1'; TextOff '0'; TextList "013016_DECIMAL_POINTS_REMOTE_DISPLAY"
      ProcessValue <- "WP231PR_DB_DR13_DEC_POINT_REM_DISPLAY"
      Visibility <- "WP231PR_DB_DR13_RS485_PROTOCOL"
   TextField "OBJECT_3" at 195,255 size 148x29; Text 'Anzahl Stopbits / Stop bits / Stop bit / Scale name'
      Visibility <- "WP231PR_DB_DR13_RS485_PROTOCOL"
   SymbolicIOField "Symbolisches EA-Feld_6" at 350,255 size 320x31; TextOn '1'; TextOff '0'; TextList "013012_RS485_STOP_BITS"
      ProcessValue <- "WP231PR_DB_DR13_RS485_STOP_BITS"
      Visibility <- "WP231PR_DB_DR13_RS485_PROTOCOL"
   Button "Up_to Setup_5_Min_2" at 670,390 size 80x80; TextOn 'Texte / text'; TextOff 'Texte / text'; PictureOff "Home_3"
      on Release: ActivateScreen("0.0.0_Scale_View_1", 0)
   Softkey "[!Invalid!]Softkey_F6" at -140,-147 size 0x0
      on KeyDown: ActivateScreen("Menu_interfaces", 0)
   Softkey "[!Invalid!]Softkey_F5" at -140,-147 size 0x0
      on KeyDown: SetTag("S1_CMD3.i_CMD_CODE", 4013); SetTag("S1_CMD3.i_CMD_TRIGGER", 1)

screen "1.5.9_DR14_S7_Interface_Parameter" 800x480, template "Template_1"
   TextField "OBJECT_33" at 0,0 size 554x34; Text '1.5.9 Einstellungen Simatic Schnittstelle / 1.5.9 Simatic Interface Settings / 1.5.9 Paramètres interface Simatic / Setup 1/3'
   Button "OBJECT_24" at 45,390 size 80x80; TextOn 'Texte / text'; TextOff 'Texte / text'; PictureOff "Exit"
      on Release: ActivateScreen("1.5.0.2_Menu_communication_interfaces_2", 0)
   Button "OBJECT_1" at 360,390 size 80x80; TextOn 'Texte / text'; TextOff 'Texte / text'; PictureOff "Save"
      on Press: SetTag("WP231PR_DB_s_CMD2_i_CMD_CODE", '4014'); SetBit("WP231PR_DB_s_CMD2_bo_CMD_TRIGGER")
   TextField "OBJECT_306" at 35,160 size 289x32; Text 'Auswahl Prozesswert 1 / Definition "Process value 1" / Sélection valeur processus 1 / Scale name'
   TextField "OBJECT_2" at 35,246 size 289x32; Text 'Auswahl Prozesswert 2 / Definition "Process value 2" / Sélection valeur processus 2 / Scale name'
   SymbolicIOField "Symbolisches EA-Feld_1" at 334,159 size 428x34; TextOn '1'; TextOff '0'; TextList "014008_SELECTION_PROC_VAL_1_S7"
      ProcessValue <- "WP231PR_DB_DR14_SEL_PROC_VAL_1_SIMATIC"
   SymbolicIOField "Symbolisches EA-Feld_2" at 335,244 size 430x34; TextOn '1'; TextOff '0'; TextList "014010_SELECTION_PROC_VAL_2_S7"
      ProcessValue <- "WP231PR_DB_DR14_SEL_PROC_VAL_2_SIMATIC"
   Button "Up_to Setup_5_Min_2" at 682,390 size 80x80; TextOn 'Texte / text'; TextOff 'Texte / text'; PictureOff "Home_3"
      on Release: ActivateScreen("0.0.0_Scale_View_1", 0)
   Softkey "[!Invalid!]Softkey_F6" at -140,-147 size 0x0
      on KeyDown: ActivateScreen("Menu_interfaces", 0)
   Softkey "[!Invalid!]Softkey_F5" at -140,-147 size 0x0
      on KeyDown: SetTag("S1_CMD3.i_CMD_CODE", 4014); SetTag("S1_CMD3.i_CMD_TRIGGER", 1)

screen "1.1_Recalibration" 800x480, template "Template_1"
   TextField "OBJECT_35" at 0,2 size 510x34; Text '1.1.1 Mit Gewichten Nachjustieren / 1.1 Recalibration / 1.1.1 Réétalonnage avec poids étalon / Calibration'
   Button "Exit to Service" at 45,390 size 80x80; TextOn 'Texte / text'; TextOff 'Texte / text'; PictureOff "Exit"
      on Release: ActivateScreen("1.0_Menu_setup", 0); SetTag("WP231PR_DB_CMD_A", 2034)
      on Press: SetTag("WP231PR_DB_s_CMD2_i_CMD_CODE", '2'); SetBit("WP231PR_DB_s_CMD2_bo_CMD_TRIGGER"); SetTag("WP231PR_DB_CMD_B", 0)
   Group "Group" at 700,5 size 95x30; Text 'Service'; PictureList "Signal_grey_yellow"
   Button "Up_to Setup_5_Min_01" at 545,390 size 80x80; TextOn 'Texte / text'; TextOff 'Texte / text'; PictureOff "Left"
      on Release: SetTag("WP231PR_DB_CMD_A", 2034)
      on Press: ActivateScreen("0.0.0_Service_Recalibration", 0); SetTag("WP231PR_DB_CMD_B", 0)
   Button "Up_to Setup_5_Min_2" at 360,390 size 80x80; TextOn 'Texte / text'; TextOff 'Texte / text'; PictureOff "Home_3"
      on Release: ActivateScreen("0.0.0_Scale_View_1", 0); SetTag("WP231PR_DB_CMD_A", 2034)
      on Press: SetTag("WP231PR_DB_s_CMD2_i_CMD_CODE", '2'); SetBit("WP231PR_DB_s_CMD2_bo_CMD_TRIGGER"); SetTag("WP231PR_DB_CMD_B", 0)
   IOField "OBJECT_301" at 0,41 size 800x90; FormatPattern ????????????????
      ProcessValue <- "WP231PR_DB_DR34_ASCII_DISPLAY"
   Button "OBJECT_28" at 110,133 size 580x70; TextOn 'Texte / text'; TextOff 'Justagegewicht 0 setzen / Set Calibration Weight 0 / Placez le poids étalon 0 / Acknowledge Empty Bin'
      on Press: SetTag("WP231PR_DB_s_CMD2_i_CMD_CODE", '60'); SetBit("WP231PR_DB_s_CMD2_bo_CMD_TRIGGER")
   Button "OBJECT_31" at 110,204 size 580x70; TextOn 'Texte / text'; TextOff 'Justagegewicht 1 setzen / Set Calibration Weight 1 / Placez le poids étalon 1 / Put & Acknowledge Calibration Weight'
      on Press: SetTag("WP231PR_DB_s_CMD2_i_CMD_CODE", '61'); SetBit("WP231PR_DB_s_CMD2_bo_CMD_TRIGGER")
   Button "OBJECT_3" at 110,276 size 580x70; TextOn 'Texte / text'; TextOff 'Justagegewicht 2 setzen (optional) / Set Calibration Weight 2 (optional) / Placez le poids étalon 2 (option) / Put & Acknowledge Calibration Weight'
      on Press: SetTag("WP231PR_DB_s_CMD2_i_CMD_CODE", '62'); SetBit("WP231PR_DB_s_CMD2_bo_CMD_TRIGGER")
   Button "Schaltfläche_1" at 670,390 size 80x80; TextOn 'Texte'; TextOff 'Texte'; PictureOff "Q_Mark"
      on Press: SetBit("S1_SHOW_HELP")
   TextField "OBJECT_4" at 210,352 size 207x32; Text 'Aktuelle Digits ADC: / Current ADC digits: / Valeur CAN / Error occurred'
      Visibility <- "S1_SHOW_HELP"
   IOField "I/O field_5" at 442,351 size 136x32; FormatPattern 9999999999
      ProcessValue <- "WP231PR_DB_DR31_DIGITS_FILTERED"
      Visibility <- "S1_SHOW_HELP"
   Softkey "[!Invalid!]Softkey_F6" at -140,-147 size 0x0
      on KeyDown: ActivateScreen("1.0_Menu_setup", 0)
   GraphicIOField "OBJECT_19" at 765,5 size 30x30; PictureList "Signal_grey_yellow"
      ProcessValue <- "WP231PR_DB_s_IO_DATA_SCALE_STATUS_2_SERVICE_MODE"
   TextField "OBJECT_37" at 700,7 size 57x25; Text 'Service / Error occurred'
   Rectangle "Rechteck_1" at 0,131 size 799x348
      Visibility <- "S1_SHOW_HELP"
   TextField "OBJECT_2" at 73,165 size 334x47; Text 'Justagegewicht 0: / Calibration weight 0: / Poids étalon 0: / Calibration'
      Visibility <- "S1_SHOW_HELP"
   TextField "OBJECT_1" at 73,230 size 334x47; Text 'Justagegewicht 1: / Calibration weight 1: / Poids étalon 1: / Calibration'
      Visibility <- "S1_SHOW_HELP"
   IOField "I/O field_1" at 415,230 size 166x47; FormatPattern 99999.99
      ProcessValue <- "WP231PR_DB_DR03_CALIB_WEIGHT_1"
      Visibility <- "S1_SHOW_HELP"
   IOField "I/O field_2" at 571,230 size 134x47; FormatPattern ????
      ProcessValue <- "WP231PR_DB_DR03_WEIGHT_UNIT"
      Visibility <- "S1_SHOW_HELP"
   IOField "I/O field_3" at 415,165 size 166x47; FormatPattern 99999.99
      ProcessValue <- "WP231PR_DB_DR03_CALIB_WEIGHT_0"
      Visibility <- "S1_SHOW_HELP"
   IOField "I/O field_4" at 571,165 size 134x47; FormatPattern ????
      ProcessValue <- "WP231PR_DB_DR03_WEIGHT_UNIT"
      Visibility <- "S1_SHOW_HELP"
   TextField "OBJECT_5" at 73,300 size 334x47; Text 'Justagegewicht 2: / Calibration weight 2: / Poids étalon 2: / Calibration'
      Visibility <- "S1_SHOW_HELP"
   IOField "I/O field_6" at 415,300 size 166x47; FormatPattern 99999.99
      ProcessValue <- "WP231PR_DB_DR03_CALIB_WEIGHT_2"
      Visibility <- "S1_SHOW_HELP"
   IOField "I/O field_7" at 571,300 size 134x47; FormatPattern ????
      ProcessValue <- "WP231PR_DB_DR03_WEIGHT_UNIT"
      Visibility <- "S1_SHOW_HELP"
   Button "Schaltfläche_2" at 642,420 size 150x50; TextOn 'Texte'; TextOff 'OK'
      on Press: ResetBit("S1_SHOW_HELP")
      Visibility <- "S1_SHOW_HELP"

screen "1.5.3_DR16_Weight_Simulation" 800x480, template "Template_1"
   TextField "OBJECT_33" at 0,0 size 356x34; Text '1.5.3 Gewichtssimulation / 1.5.3 Weightsimulation / 1.5.3 Simulation poids / Setup 2/3'
   Button "OBJECT_24" at 45,390 size 80x80; TextOn 'Texte / text'; TextOff 'Texte / text'; PictureOff "Exit"
      on Release: SetTag("WP231PR_DB_CMD_B", 0)
      on Press: ActivateScreen("1.5.0.1_Menu_communication_interfaces_1", 0); SetTag("WP231PR_DB_CMD_A", 2035)
   TextField "OBJECT_10" at 9,93 size 245x29; Text 'Zu simulierendes Gewicht / Weight to simulate / Poids à simuler / Display Resolution'
   IOField "OBJECT_4" at 258,82 size 222x50; FormatPattern 999999.9999
      ProcessValue <- "WP231PR_DB_DR16_SIMULATION_WEIGHT"
   IOField "I/O field_2" at 482,83 size 60x50; FormatPattern ????
      ProcessValue <- "WP231PR_DB_DR03_WEIGHT_UNIT"
   Button "OBJECT_28" at 95,143 size 290x70; TextOn 'Texte / text'; TextOff 'Start Simulation / Démarrer la simulation / Acknowledge Empty Bin'
      on Release: SetTag("WP231PR_DB_s_CMD2_i_CMD_CODE", '3'); SetBit("WP231PR_DB_s_CMD2_bo_CMD_TRIGGER")
      on Press: SetTag("WP231PR_DB_s_CMD1_i_CMD_CODE", 4016); SetBit("WP231PR_DB_s_CMD1_bo_CMD_TRIGGER")
   Button "OBJECT_2" at 416,143 size 290x70; TextOn 'Texte / text'; TextOff 'Stop Simulation / Arrêt simulation / Acknowledge Empty Bin'
      on Press: SetTag("WP231PR_DB_s_CMD2_i_CMD_CODE", '4'); SetBit("WP231PR_DB_s_CMD2_bo_CMD_TRIGGER")
   GraphicIOField "OBJECT_45" at 765,5 size 30x30; PictureList "Signal_grey_green"
      ProcessValue <- "WP231PR_DB_s_IO_DATA_SCALE_STATUS_2_SIMULATION_MODE"
   TextField "OBJECT_53" at 678,8 size 81x25; Text 'Simulation / simulation / Error occurred'
   TextField "OBJECT_6" at 11,214 size 151x28; Text 'Digitale Eingänge / Digital Inputs / Entrées TOR / Scale name'
   TextField "OBJECT_7" at 7,247 size 75x27; Text 'DI.0 / Entrée 0 / Scale name'
   TextField "OBJECT_8" at 7,279 size 75x27; Text 'DI.1 / Entrée 1 / Scale name'
   TextField "OBJECT_1" at 7,312 size 75x27; Text 'DI.2 / Entrée 2 / Scale name'
   TextField "OBJECT_11" at 7,342 size 75x27; Text 'DI.3 / Entrée 3 / Scale name'
   TextField "OBJECT_12" at 214,245 size 68x27; Text 'DQ.0 / Sortie 0 / Scale name'
   TextField "OBJECT_13" at 214,311 size 68x27; Text 'DQ.2 / Sortie 2 / Scale name'
   TextField "OBJECT_14" at 214,278 size 68x27; Text 'DQ.1 / Sortie 1 / Scale name'
   TextField "OBJECT_15" at 214,345 size 68x27; Text 'DQ.3 / Sortie 3 / Scale name'
   GraphicIOField "OBJECT_304" at 89,246 size 40x30; PictureList "Signal_grey_yellow"
      ProcessValue <- "WP231PR_DB_DR31_CURRENT_STATE_DI_0"
   GraphicIOField "OBJECT_16" at 89,279 size 40x30; PictureList "Signal_grey_yellow"
      ProcessValue <- "WP231PR_DB_DR31_CURRENT_STATE_DI_1"
   GraphicIOField "OBJECT_17" at 89,312 size 40x30; PictureList "Signal_grey_yellow"
      ProcessValue <- "WP231PR_DB_DR31_CURRENT_STATE_DI_2"
   GraphicIOField "OBJECT_18" at 89,346 size 40x30; PictureList "Signal_grey_yellow"
      ProcessValue <- "WP231PR_DB_DR31_CURRENT_STATE_DI_3"
   GraphicIOField "OBJECT_19" at 289,246 size 40x30; PictureList "Signal_grey_yellow"
      ProcessValue <- "WP231PR_DB_DR31_CURRENT_STATE_DQ_0"
   GraphicIOField "OBJECT_20" at 289,312 size 40x30; PictureList "Signal_grey_yellow"
      ProcessValue <- "WP231PR_DB_DR31_CURRENT_STATE_DQ_2"
   GraphicIOField "OBJECT_21" at 289,279 size 40x30; PictureList "Signal_grey_yellow"
      ProcessValue <- "WP231PR_DB_DR31_CURRENT_STATE_DQ_1"
   GraphicIOField "OBJECT_22" at 289,346 size 40x30; PictureList "Signal_grey_yellow"
      ProcessValue <- "WP231PR_DB_DR31_CURRENT_STATE_DQ_3"
   TextField "OBJECT_3" at 205,214 size 155x28; Text 'Digitale Ausgänge / Digital Outputs / Sorties TOR / Scale name'
   IOField "OBJECT_9" at 489,297 size 63x30; FormatPattern 99999
      ProcessValue <- "WP231PR_DB_DR31_CURRENT_ANA_OUT_DIGITS"
   TextField "OBJECT_5" at 429,214 size 150x28; Text 'Analogausgang / Analogue out / Sortie analogique / Scale name'
   GraphicIOField "OBJECT_23" at 713,246 size 40x30; PictureList "Signal_grey_yellow"
      ProcessValue <- "WP231PR_DB_s_IO_DATA_SCALE_STATUS_1_LIMIT_1"
   TextField "OBJECT_25" at 610,214 size 100x28; Text 'Grenzwerte / Limits / Limites / Error occurred'
   TextField "OBJECT_26" at 607,247 size 99x26; Text 'Grenzwert 1 / Limit 1 / Limite 1 / Error occurred'
   GraphicIOField "OBJECT_31" at 713,279 size 40x30; PictureList "Signal_grey_yellow"
      ProcessValue <- "WP231PR_DB_s_IO_DATA_SCALE_STATUS_1_LIMIT_2"
   TextField "OBJECT_27" at 608,279 size 99x26; Text 'Grenzwert 2 / Limit 2 / Limite 2 / Error occurred'
   Bar "Balken_1" at 449,251 size 36x129; MinimumValue 0; MaximumValue 65535
      ProcessValue <- "WP231PR_DB_DR31_CURRENT_ANA_OUT_DIGITS"
   TextField "Textfeld_2" at 509,360 size 43x25; Text '0 mA / 0mA'
   TextField "Textfeld_3" at 510,244 size 52x25; Text '24 mA / 24mA'
   TextField "Textfeld_4" at 555,299 size 44x25; Text 'digits'
   IOField "OBJECT_301" at 0,40 size 800x40; FormatPattern ????????????????
      ProcessValue <- "WP231PR_DB_DR34_ASCII_DISPLAY"
   Softkey "[!Invalid!]Softkey_F6" at -140,-147 size 0x0
      on KeyDown: ActivateScreen("1.5.0.1_Menu_communication_interfaces_1", 0)
   Group "Group" at 0,33 size 800x352; Text 'Die Gewichtssimulation ist zur Zeit nicht freigeschaltet. Bitte gehen Sie zu "1.4.3 Erweiterte Waagenparameter" und schalten Sie die Funktion frei.'
   Rectangle "Rechteck_1" at 0,33 size 800x352
      Visibility <- "WP231PR_DB_DR03_WEIGHT_SIM_ALLOWED"
   TextField "Textfeld_1" at 37,71 size 763x116; Text 'Die Gewichtssimulation ist zur Zeit nicht freigeschaltet. Bitte gehen Sie zu "1.4.3 Erweiterte Waagenparameter" und schalten Sie die Funktion frei. Weight Simulation is disabled at the moment! Please go to "1.4.3 Advanced Scale Parameter" and enable it. La simulation du poids n'est pas possible. Voir le point 1.4.3 et libérer la fonction'
      Visibility <- "WP231PR_DB_DR03_WEIGHT_SIM_ALLOWED"

screen "1.5.1.2_DR7_digital_in_outputs_2" 800x480, template "Template_1"
   TextField "OBJECT_33" at 0,0 size 766x34; Text '1.5.1.2 Einstellungen Digital Ein- und Ausgänge 2 von 2 / 1.5.1.2 Digital In- and Outputs Settings 2 of 2 / 1.5.1.2 Paramétrage E/S TOR 2/2 / Setup 1/3'
   TextField "OBJECT_9" at 290,56 size 335x30; Text 'Funktionszuweisung / Functions for Digital Outputs / Affectation de la fonction / Scale name'
   TextField "OBJECT_11" at 5,96 size 164x34; Text 'Ausgang DQ.0 / Output DQ.0 / Sortie TOR 0 / Scale name'
   TextField "OBJECT_12" at 5,219 size 164x34; Text 'Ausgang DQ.2 / Output DQ.2 / Sortie TOR 2 / Weight Unit'
   TextField "OBJECT_13" at 5,277 size 164x34; Text 'Ausgang DQ.3 / Output DQ.3 / Sortie TOR 3 / Weight Unit'
   TextField "OBJECT_14" at 5,159 size 164x34; Text 'Ausgang DQ.1 / Output DQ.1 / Sortie TOR 1 / Scale name'
   SymbolicIOField "Symbolisches EA-Feld_1" at 289,96 size 360x36; TextOn '1'; TextOff '0'; TextList "007020_ASSIGNMENT_DIGITAL_OUTPUT"
      ProcessValue <- "WP231PR_DB_DR07_ASSIGN_DQ_0"
   SymbolicIOField "Symbolisches EA-Feld_2" at 289,159 size 360x36; TextOn '1'; TextOff '0'; TextList "007020_ASSIGNMENT_DIGITAL_OUTPUT"
      ProcessValue <- "WP231PR_DB_DR07_ASSIGN_DQ_1"
   SymbolicIOField "Symbolisches EA-Feld_3" at 289,219 size 360x36; TextOn '1'; TextOff '0'; TextList "007020_ASSIGNMENT_DIGITAL_OUTPUT"
      ProcessValue <- "WP231PR_DB_DR07_ASSIGN_DQ_2"
   SymbolicIOField "Symbolisches EA-Feld_4" at 289,277 size 360x36; TextOn '1'; TextOff '0'; TextList "007020_ASSIGNMENT_DIGITAL_OUTPUT"
      ProcessValue <- "WP231PR_DB_DR07_ASSIGN_DQ_3"
   Button "Up_to Setup_5_Min_01" at 545,390 size 80x80; TextOn 'Texte / text'; TextOff 'Texte / text'; PictureOff "Left"
      on Release: ActivateScreen("1.5.1.1_DR7_digital_in_outputs_1", 0)
   Button "OBJECT_24" at 45,390 size 80x80; TextOn 'Texte / text'; TextOff 'Texte / text'; PictureOff "Exit"
      on Release: ActivateScreen("1.5.0.1_Menu_communication_interfaces_1", 0)
   SymbolicIOField "Symbolisches EA-Feld_5" at 289,336 size 361x36; TextOn '1'; TextOff '0'; TextList "007026_DIGIT_STATUS_BY_ERROR_STOP"
      ProcessValue <- "WP231PR_DB_DR07_ANA_OUT_BY_ERR_OR_STOP"
   TextField "OBJECT_1" at 5,336 size 275x34; Text 'Störungs-Stop-Verhalten / Error-Stop-Status / Erreur - Stop / Weight Unit'
   SymbolicIOField "Symbolisches EA-Feld_6" at 668,97 size 118x36; TextOn '1'; TextOff '0'; TextList "003072_FALSE_TRUE"
      ProcessValue <- "WP231PR_DB_DR07_DQ_0_BY_ERR_OR_STOP"
      Visibility <- "WP231PR_DB_DR07_ANA_OUT_BY_ERR_OR_STOP"
   SymbolicIOField "Symbolisches EA-Feld_7" at 668,162 size 118x36; TextOn '1'; TextOff '0'; TextList "003072_FALSE_TRUE"
      ProcessValue <- "WP231PR_DB_DR07_DQ_1_BY_ERR_OR_STOP"
      Visibility <- "WP231PR_DB_DR07_ANA_OUT_BY_ERR_OR_STOP"
   SymbolicIOField "Symbolisches EA-Feld_8" at 668,220 size 118x36; TextOn '1'; TextOff '0'; TextList "003072_FALSE_TRUE"
      ProcessValue <- "WP231PR_DB_DR07_DQ_2_BY_ERR_OR_STOP"
      Visibility <- "WP231PR_DB_DR07_ANA_OUT_BY_ERR_OR_STOP"
   SymbolicIOField "Symbolisches EA-Feld_9" at 668,278 size 120x36; TextOn '1'; TextOff '0'; TextList "003072_FALSE_TRUE"
      ProcessValue <- "WP231PR_DB_DR07_DQ_3_BY_ERR_OR_STOP"
      Visibility <- "WP231PR_DB_DR07_ANA_OUT_BY_ERR_OR_STOP"
   Button "OBJECT_3" at 360,390 size 80x80; TextOn 'Texte / text'; TextOff 'Texte / text'; PictureOff "Save"
      on Press: SetTag("WP231PR_DB_s_CMD2_i_CMD_CODE", '4007'); SetBit("WP231PR_DB_s_CMD2_bo_CMD_TRIGGER")
   TextField "Textfeld_1" at 660,57 size 130x30; Text 'Ersatzwert / Error/Stop status / Valeur'
      Visibility <- "WP231PR_DB_DR07_ANA_OUT_BY_ERR_OR_STOP"
   Softkey "[!Invalid!]Softkey_F6" at -140,-147 size 0x0
      on KeyDown: ActivateScreen("1.5.0.1_Menu_communication_interfaces_1", 0)
   Softkey "[!Invalid!]Softkey_F5" at -140,-147 size 0x0
      on KeyDown: ActivateScreen("DR7_Process_Interfaces_3", 0)
   Softkey "[!Invalid!]Softkey_F4" at -140,-147 size 0x0
      on KeyDown: ActivateScreen("1.5.1.1_DR7_digital_in_outputs_1", 0)

screen "2.5.1_Trace_Start_Stop" 800x480, template "Template_1"
   TextField "OBJECT_33" at 0,0 size 397x34; Text '2.5.1 Trace Start / Stop / 2.6.1 Démarrer/arrêter trace / Setup 2/3'
   Button "OBJECT_24" at 45,390 size 80x80; TextOn 'Texte / text'; TextOff 'Texte / text'; PictureOff "Exit"
      on Release: ActivateScreen("2.0_Menu_diagnostic", 0)
   GraphicIOField "OBJECT_18" at 765,5 size 30x30; PictureList "Signal_grey_green"
      ProcessValue <- "WP231PR_DB_s_IO_DATA_SCALE_STATUS_2_TRACE"
   TextField "OBJECT_57" at 716,7 size 46x25; Text 'Trace / trace / Error occurred'
   Button "OBJECT_1" at 33,104 size 350x90; TextOn 'Texte / text'; TextOff 'Start Trace / Démarrer Trace / Acknowledge Empty Bin'
      on Release: SetTag("WP231PR_DB_s_CMD2_i_CMD_CODE", '451'); SetBit("WP231PR_DB_s_CMD2_bo_CMD_TRIGGER")
   Button "OBJECT_4" at 416,104 size 350x90; TextOn 'Texte / text'; TextOff 'Stop Trace / Arrêt trace / Acknowledge Empty Bin'
      on Release: SetTag("WP231PR_DB_s_CMD2_i_CMD_CODE", '452'); SetBit("WP231PR_DB_s_CMD2_bo_CMD_TRIGGER")
   Button "Schaltfläche_1" at 670,390 size 80x80; TextOn 'Texte'; TextOff 'Texte'; PictureOff "Q_Mark"
      on Press: SetBit("S1_SHOW_HELP")
   Button "OBJECT_2" at 33,244 size 350x90; TextOn 'Texte / text'; TextOff 'Einzel-Trace-Element / Single Trace / Trace une fois / Acknowledge Empty Bin'
      on Release: SetTag("WP231PR_DB_s_CMD2_i_CMD_CODE", '453'); SetBit("WP231PR_DB_s_CMD2_bo_CMD_TRIGGER")
   Button "OBJECT_3" at 416,244 size 350x90; TextOn 'Texte / text'; TextOff 'Trace Speicher löschen / Delete Trace Memory / Effacer mémoire trace / Acknowledge Empty Bin'
      on Release: SetTag("WP231PR_DB_s_CMD2_i_CMD_CODE", '454'); SetBit("WP231PR_DB_s_CMD2_bo_CMD_TRIGGER")
   Softkey "[!Invalid!]Softkey_F6" at -140,-147 size 0x0
      on KeyDown: ActivateScreen("2.0_Menu_diagnostic", 0)
   TextField "Textfeld_1" at 0,57 size 800x422; Text 'Die Tracefunktion der Baugruppe ermöglicht es alle waageninternen Prozesswerte wie Gewicht, E/A Status usw. mit einem Aufzeichnungszyklus von bis zu 10ms aufzuzeichnen. Die Funktion dient der Inbetriebnahme, der Optimierung und der Fehlersuche. Der Trace-Rekorder soll im Normalbetrieb nicht aktiv sein. Die aufgezeichneten Daten können nur mittels eines PC und der Software "SIWATOOL V7" ausgelesen werden! The trace functionality provides a record of all scale internal process values like the weight, I/O status etc. with a recording cycle down to 10ms. This recorder can be used for commissioning, optimizing and trouble shooting. The Trace-Recorder should not be running in normal operation. The recorded data can be read only with a PC and "SIWATOOL V7" software! La fonction trace pour visualiser toutes les valeurs'
      Visibility <- "S1_SHOW_HELP"
   Button "Schaltfläche_2" at 643,423 size 150x50; TextOn 'Texte'; TextOff 'OK'
      on Press: ResetBit("S1_SHOW_HELP")
      Visibility <- "S1_SHOW_HELP"

screen "1.5.0.1_Menu_communication_interfaces_1" 800x480, template "Template_1"
   TextField "OBJECT_82" at 0,0 size 709x34; Text '1.5.0 Kommunikation & Schnittstellen Seite 1 von 2 / 1.5.0 Communication & Interfaces 1 of 2 / 1.5.0 Communication et Interfaces 1/2 / Main Menu'
   Button "Exit_to_Main_menue" at 45,390 size 80x80; TextOn 'Texte / text'; TextOff 'Texte / text'; PictureOff "Exit"
      on Press: ActivateScreen("1.0_Menu_setup", 0)
   Button "Exit_to_Main_menue_1" at 670,390 size 80x80; TextOn 'Texte / text'; TextOff 'Texte / text'; PictureOff "Right"
      on Press: ActivateScreen("1.5.0.2_Menu_communication_interfaces_2", 0)
   Button "Password" at 416,73 size 350x90; TextOn 'Texte / text'; TextOff '1.5.4 Test & Steuern Digital-Ausgänge 1.5.4 Test & Force Digital Outputs 1.5.4 Test & contrôle des E/S TOR Diagnostics'
      on Release: ActivateScreen("1.5.4_DR18_control_digital_outputs", 0); SetTag("WP231PR_DB_CMD_B", 2031)
      on Press: SetTag("WP231PR_DB_s_CMD2_i_CMD_CODE", '2018'); SetTag("WP231PR_DB_s_CMD1_i_CMD_CODE", '2007'); SetBit("WP231PR_DB_s_CMD2_bo_CMD_TRIGGER")
   Button "Expert calibration" at 33,73 size 350x90; TextOn 'Texte / text'; TextOff '1.5.1 Einstellungen Digital Ein- & Ausgänge 1.5.1 Digital In- and Output 1.5.1 Paramétrage E/S TOR Enhanced Scale Setup'
      on Press: SetTag("WP231PR_DB_s_CMD1_i_CMD_CODE", '2007'); SetBit("WP231PR_DB_s_CMD1_bo_CMD_TRIGGER")
      on Release: ActivateScreen("1.5.1.1_DR7_digital_in_outputs_1", 0)
   Button "Expert calibration_1" at 33,174 size 350x90; TextOn 'Texte / text'; TextOff '1.5.2 Einstellungen Analogausgang 1.5.2 Analogue Output 1.5.2 Paramétrage sortie analogique Enhanced Scale Setup'
      on Release: ActivateScreen("1.5.2_DR7_Analogue_Output", 0)
      on Press: SetTag("WP231PR_DB_s_CMD2_i_CMD_CODE", '2007'); SetBit("WP231PR_DB_s_CMD2_bo_CMD_TRIGGER")
   Button "OBJECT_3" at 416,174 size 350x90; TextOn 'Texte / text'; TextOff '1.5.5 Test & Steuern Analog-Ausgang 1.5.5 Test & Force Analogue Output 1.5.5 Test & contrôle sortie analogique Quick Scale Setup'
      on Release: ActivateScreen("1.5.5_DR17_control_analogue_output", 0); SetTag("WP231PR_DB_s_CMD2_i_CMD_CODE", '2007'); SetBit("WP231PR_DB_s_CMD2_bo_CMD_TRIGGER")
      on Press: SetTag("WP231PR_DB_s_CMD1_i_CMD_CODE", '2017'); SetBit("WP231PR_DB_s_CMD1_bo_CMD_TRIGGER")
   Button "Expert calibration_2" at 33,275 size 350x90; TextOn 'Texte / text'; TextOff '1.5.3 Gewichtssimulation / 1.5.3 Weight Simulation / 1.5.3 Simulation poids / Enhanced Scale Setup'
      on Release: ActivateScreen("1.5.3_DR16_Weight_Simulation", 0); SetTag("WP231PR_DB_CMD_B", 2031); SetTag("WP231PR_DB_CMD_A", 2034)
      on Press: SetTag("WP231PR_DB_s_CMD2_i_CMD_CODE", '2016'); SetBit("WP231PR_DB_s_CMD2_bo_CMD_TRIGGER")
   Button "Expert calibration_3" at 416,275 size 350x90; TextOn 'Texte / text'; TextOff '1.5.6 Einstellungen RS485 / 1.5.6 RS485 Settings / 1.5.6 Paramétrage RS485 / Enhanced Scale Setup'
      on Press: SetTag("WP231PR_DB_s_CMD2_i_CMD_CODE", '2013'); SetBit("WP231PR_DB_s_CMD2_bo_CMD_TRIGGER")
      on Release: ActivateScreen("1.5.6_DR13_RS485-Parameter", 0)
   Softkey "[!Invalid!]Softkey_F6" at -140,-147 size 0x0
      on KeyDown: ActivateScreen("1.0_Menu_setup", 0)

screen "1.0_Menu_setup" 800x480, template "Template_1"
   TextField "OBJECT_82" at 0,0 size 262x34; Text '1.0 Setup / 1.0 Mise en service / Main Menu'
   Button "Expert calibration" at 416,73 size 350x90; TextOn 'Texte / text'; TextOff '1.4 Erweiterte Waagenparameter 1.4 Advanced Scale Parameters 1.4 Tous les paramètres Enhanced Scale Setup'
      on Press: ActivateScreen("0.0.0_Service_Adv_Scale_Para", 0)
   Button "Exit_to_Main_menue" at 45,390 size 80x80; TextOn 'Texte / text'; TextOff 'Texte / text'; PictureOff "Exit"
      on Release: ActivateScreen("0.0.0_Menu_main", 0)
   Button "Recalibration" at 33,73 size 350x90; TextOn 'Texte / text'; TextOff '1.1 Nachjustage / 1.1 Recalibration / 1.1 Réétalonnage / Module Info'
      on Release: SetTag("WP231PR_DB_CMD_A", 2034)
      on Press: ActivateScreen("0.0.0_Service_Recalibration", 0); SetTag("WP231PR_DB_CMD_B", 2031)
   Button "Recalibration_1" at 416,275 size 350x90; TextOn 'Texte / text'; TextOff '1.6 Wiederherstellungs- punkt 1.6 Recovery / Reset 1.6 Point de sauvegarde Module Info'
      on Press: ActivateScreen("0.0.0_Service_Recovery", 0)
   Group "Group" at 700,5 size 95x30; Text 'Service'; PictureList "Signal_grey_yellow"
   Button "5-Minute_Setup" at 33,277 size 350x90; TextOn 'Texte / text'; TextOff '1.3 Grenzwerte / 1.3 Limits / 1.3 Limites / Quick Scale Setup'
      on Release: SetTag("WP231PR_DB_s_CMD2_i_CMD_CODE", 2003); SetBit("WP231PR_DB_s_CMD2_bo_CMD_TRIGGER"); ActivateScreen("1.3.1_DR6_ Limit_values", 0)
      on Press: SetTag("WP231PR_DB_s_CMD1_i_CMD_CODE", 2006); SetBit("WP231PR_DB_s_CMD1_bo_CMD_TRIGGER")
   Button "5-Minute_Setup_1" at 33,174 size 350x90; TextOn 'Texte / text'; TextOff '1.2 Quick Start / 1.2 Mise en service rapide / Quick Scale Setup'
      on Press: ActivateScreen("0.0.0_Service_Quick_Start", 0)
   Button "Expert settings" at 416,174 size 350x90; TextOn 'Texte / text'; TextOff '1.5 Kommunikation & Schnittstellen 1.5 Communication & Interfaces 1.5 Communication et interfaces Enhanced Scale Setup'
      on Release: ActivateScreen("1.5.0.1_Menu_communication_interfaces_1", 0)
   Softkey "[!Invalid!]Softkey_F6" at -140,-147 size 0x0
      on KeyDown: SetTag("S1_CMD2.i_CMD_CODE", 2); SetTag("S1_CMD2.i_CMD_TRIGGER", 1); ActivateScreen("0.0.0_Menu_main", 0)
   GraphicIOField "OBJECT_19" at 765,5 size 30x30; PictureList "Signal_grey_yellow"
      ProcessValue <- "WP231PR_DB_s_IO_DATA_SCALE_STATUS_2_SERVICE_MODE"
   TextField "OBJECT_37" at 700,7 size 57x25; Text 'Service / Error occurred'

screen "1.6.1_Recovery_point" 800x480, template "Template_1"
   TextField "OBJECT_33" at 0,0 size 425x34; Text '1.6.1 Wiederherstellungspunkt / 1.6.1 Recovery Point / 1.6.1 Point de sauvegarde / Setup 2/3'
   Button "OBJECT_24" at 45,390 size 80x80; TextOn 'Texte / text'; TextOff 'Texte / text'; PictureOff "Exit"
      on Release: ActivateScreen("1.0_Menu_setup", 0)
      on Press: SetTag("WP231PR_DB_s_CMD2_i_CMD_CODE", '2'); SetBit("WP231PR_DB_s_CMD2_bo_CMD_TRIGGER")
   Button "OBJECT_28" at 33,73 size 350x90; TextOn 'Texte / text'; TextOff 'Wiederherstellungspunkt erstellen Create Recovery Point Créer un point de sauvegarde Acknowledge Empty Bin'
      on Release: SetTag("WP231PR_DB_s_CMD2_i_CMD_CODE", '51'); SetBit("WP231PR_DB_s_CMD2_bo_CMD_TRIGGER")
   Button "OBJECT_2" at 33,174 size 350x90; TextOn 'Texte / text'; TextOff 'Wiederherstellungspunkt laden Load Recovery Point Recharger un point de sauvegarde Acknowledge Empty Bin'
      on Release: SetTag("WP231PR_DB_s_CMD2_i_CMD_CODE", '31'); SetBit("WP231PR_DB_s_CMD2_bo_CMD_TRIGGER")
   Button "OBJECT_1" at 416,73 size 350x90; TextOn 'Texte / text'; TextOff 'Werkseinstellungen laden Load Factory Settings Recharger les paramètres usines Acknowledge Empty Bin'
      on Release: SetTag("WP231PR_DB_s_CMD2_i_CMD_CODE", '11'); SetBit("WP231PR_DB_s_CMD2_bo_CMD_TRIGGER")
   Button "OBJECT_3" at 33,275 size 350x90; TextOn 'Texte / text'; TextOff 'Standard Wägeparameter laden Load Standard Scale Parameter Paramètres standards Acknowledge Empty Bin'
      on Release: SetTag("WP231PR_DB_s_CMD2_i_CMD_CODE", '12'); SetBit("WP231PR_DB_s_CMD2_bo_CMD_TRIGGER")
   Group "Group" at 700,5 size 95x30; Text 'Service'; PictureList "Signal_grey_yellow"
   Button "Schaltfläche_1" at 670,390 size 80x80; TextOn 'Texte'; TextOff 'Texte'; PictureOff "Q_Mark"
      on Press: SetBit("S1_SHOW_HELP")
   Button "Up_to Setup_5_Min_2" at 360,390 size 80x80; TextOn 'Texte / text'; TextOff 'Texte / text'; PictureOff "Home_3"
      on Release: ActivateScreen("0.0.0_Scale_View_1", 0)
      on Press: SetTag("WP231PR_DB_s_CMD2_i_CMD_CODE", '2'); SetBit("WP231PR_DB_s_CMD2_bo_CMD_TRIGGER")
   Softkey "[!Invalid!]Softkey_F6" at -140,-147 size 0x0
      on KeyDown: ActivateScreen("1.0_Menu_setup", 0)
   GraphicIOField "OBJECT_19" at 765,5 size 30x30; PictureList "Signal_grey_yellow"
      ProcessValue <- "WP231PR_DB_s_IO_DATA_SCALE_STATUS_2_SIMULATION_MODE"
   TextField "OBJECT_37" at 700,7 size 57x25; Text 'Service / Error occurred'
   TextField "Textfeld_1" at 0,57 size 800x422; Text 'Nach erfolgreicher Inbetriebnahme, kann ein Wiederherstellungspunkt für die Waage erstellt werden. Dieser kann dann zu einem späteren Zeitpunkt wieder geladen werden und versetzt die Waage zurück in den Zustand direkt nach der Inbetriebnahme. Mittels "Standard Wägeparameter laden" werden bis auf die Kommunikationseinstellungen (Ethernet, RS485) alle Waagen- parameter zurück gesetzt. "Werkseinstellungen laden" setzt die Baugruppe komplett auf Werkseinstellungen zurück. After a successful commissioning, a "Recovery Point" can be created. This point can be loaded later on and sets the scale back to the state after the commissioning. Via "Load Standard Scale Parameter" besides the communication settings for the ethernet and RS485 interface, all settings are restored to factory default. Via "Load factory Settings" all parameters are restored to factory default. Point de sauvegarde après la mise en service'
      Visibility <- "S1_SHOW_HELP"
   Button "Schaltfläche_2" at 643,423 size 150x50; TextOn 'Texte'; TextOff 'OK'
      on Press: ResetBit("S1_SHOW_HELP")
      Visibility <- "S1_SHOW_HELP"

screen "0.0.0_Service_Recalibration" 800x480, template "Template_1"
   Softkey "[!Invalid!]Softkey_F6" at -140,-147 size 0x0
      on KeyDown: SetTag("S1_CMD3.i_CMD_CODE", 2); SetTag("S1_CMD3.i_CMD_TRIGGER", 1); ActivateScreen("0.0.0_Menu_main", 0); function_efd93a16()
   Softkey "[!Invalid!]Softkey_F5" at -140,-147 size 0x0
      on KeyDown: SetTag("S1_CMD3.i_CMD_CODE", 1); SetTag("S1_CMD3.i_CMD_TRIGGER", 1); ActivateScreen("1.0_Menu_setup", 0)
   TextField "OBJECT_35" at 0,0 size 336x34; Text 'Nachjustage - Warnung / Recalibration - Warning / Réétalonnage / Calibration'
   Button "OBJECT_24" at 45,390 size 80x80; TextOn 'Texte / text'; TextOff 'Texte / text'; PictureOff "Exit"
      on Release: ActivateScreen("1.0_Menu_setup", 0)
      on Press: SetTag("WP231PR_DB_s_CMD2_i_CMD_CODE", 2); SetBit("WP231PR_DB_s_CMD2_bo_CMD_TRIGGER")
   TextField "OBJECT_1" at 24,89 size 127x33; Text 'Achtung! / Warning! / Attention / Calibration'
   TextField "OBJECT_2" at 18,130 size 767x91; Text 'Für die Nachjustage muss die Waage in den Service-Betrieb geschaltet werden. Sie haben Zugriff auf alle Waagenparameter. Die aktuelle Waagenkennlinie wird überschrieben! For "Recalibration" the scale needs to be in Service Mode. You will have full access to critical parameters! The current scale curve will be overwritten! Mode service requis pour le réétalonnage Calibration'
   Button "OBJECT_34" at 670,390 size 80x80; TextOn 'Texte / text'; TextOff 'Texte / text'; PictureOff "Right"
      on Release: ActivateScreen("1.1_Recalibration", 0); SetTag("WP231PR_DB_CMD_B", 2031)
      on Press: SetTag("WP231PR_DB_s_CMD2_i_CMD_CODE", '2003'); SetTag("WP231PR_DB_s_CMD2_bo_CMD_TRIGGER", 1)
   Button "Service on_1" at 225,280 size 350x90; TextOn 'Texte / text'; TextOff 'Servicebetrieb einschalten Switch On "Service Mode" Mettre en mode service Acknowledge Empty Bin'
      on Press: SetTag("WP231PR_DB_s_CMD2_i_CMD_CODE", '1'); SetBit("WP231PR_DB_s_CMD2_bo_CMD_TRIGGER")
   Group "Group" at 700,5 size 95x30; Text 'Service'; PictureList "Signal_grey_yellow"
   GraphicIOField "OBJECT_19" at 765,5 size 30x30; PictureList "Signal_grey_yellow"
      ProcessValue <- "WP231PR_DB_s_IO_DATA_SCALE_STATUS_2_SERVICE_MODE"
   TextField "OBJECT_37" at 700,7 size 57x25; Text 'Service / Error occurred'

screen "1.5.4_DR18_control_digital_outputs" 800x480, template "Template_1"
   Softkey "[!Invalid!]Softkey_F6" at -140,-147 size 0x0
      on KeyDown: ActivateScreen("1.5.0.1_Menu_communication_interfaces_1", 0)
   SymbolicIOField "Symbolisches EA-Feld_5" at 525,100 size 200x31; TextOn '1'; TextOff '0'; TextList "FORCE_DIGITAL_IO"
      ProcessValue <- "WP231PR_DB_DR18_DEF_DIG_OUT_DQ_0"
      Visibility <- "WP231PR_DB_DR07_ASSIGN_DQ_0"
   SymbolicIOField "Symbolisches EA-Feld_6" at 525,160 size 200x31; TextOn '1'; TextOff '0'; TextList "FORCE_DIGITAL_IO"
      ProcessValue <- "WP231PR_DB_DR18_DEF_DIG_OUT_DQ_1"
      Visibility <- "WP231PR_DB_DR07_ASSIGN_DQ_1"
   SymbolicIOField "Symbolisches EA-Feld_7" at 525,220 size 200x31; TextOn '1'; TextOff '0'; TextList "FORCE_DIGITAL_IO"
      ProcessValue <- "WP231PR_DB_DR18_DEF_DIG_OUT_DQ_2"
      Visibility <- "WP231PR_DB_DR07_ASSIGN_DQ_2"
   SymbolicIOField "Symbolisches EA-Feld_8" at 525,279 size 200x31; TextOn '1'; TextOff '0'; TextList "FORCE_DIGITAL_IO"
      ProcessValue <- "WP231PR_DB_DR18_DEF_DIG_OUT_DQ_3"
      Visibility <- "WP231PR_DB_DR07_ASSIGN_DQ_3"
   TextField "OBJECT_33" at 0,0 size 492x32; Text '1.5.4 Test / Steuern Digital-Ausgänge / 1.5.4 Test / Force Digital Outputs / 1.5.4 Test & contrôle des E/S TOR / Setup 2/3'
   Button "OBJECT_24" at 45,390 size 80x80; TextOn 'Texte / text'; TextOff 'Texte / text'; PictureOff "Exit"
      on Release: ActivateScreen("1.5.0.1_Menu_communication_interfaces_1", 0); SetTag("WP231PR_DB_CMD_B", 0)
   Button "OBJECT_11" at 360,390 size 80x80; TextOn 'Texte / text'; TextOff 'Texte / text'; PictureOff "Save"
      on Release: SetTag("WP231PR_DB_s_CMD2_i_CMD_CODE", '4018'); SetBit("WP231PR_DB_s_CMD2_bo_CMD_TRIGGER")
   TextField "OBJECT_1" at 194,62 size 336x30; Text 'Aktuelle Funktionszuweisung / Functions for Digital Outputs / Afficher fonction actuelle / Scale name'
   TextField "OBJECT_2" at 5,100 size 164x34; Text 'Ausgang DQ.0 / Output DQ.0 / Sortie TOR 0 / Scale name'
   TextField "OBJECT_12" at 5,220 size 164x34; Text 'Ausgang DQ.2 / Output DQ.2 / Sortie TOR 2 / Weight Unit'
   TextField "OBJECT_13" at 5,282 size 164x34; Text 'Ausgang DQ.3 / Output DQ.3 / Sortie TOR 3 / Weight Unit'
   TextField "OBJECT_14" at 5,159 size 164x34; Text 'Ausgang DQ.1 / Output DQ.1 / Sortie TOR 1 / Scale name'
   SymbolicIOField "Symbolisches EA-Feld_1" at 184,103 size 326x28; TextOn '1'; TextOff '0'; TextList "007020_ASSIGNMENT_DIGITAL_OUTPUT"
      ProcessValue <- "WP231PR_DB_DR07_ASSIGN_DQ_0"
   SymbolicIOField "Symbolisches EA-Feld_2" at 184,161 size 326x28; TextOn '1'; TextOff '0'; TextList "007020_ASSIGNMENT_DIGITAL_OUTPUT"
      ProcessValue <- "WP231PR_DB_DR07_ASSIGN_DQ_1"
   SymbolicIOField "Symbolisches EA-Feld_3" at 184,223 size 326x28; TextOn '1'; TextOff '0'; TextList "007020_ASSIGNMENT_DIGITAL_OUTPUT"
      ProcessValue <- "WP231PR_DB_DR07_ASSIGN_DQ_2"
   SymbolicIOField "Symbolisches EA-Feld_4" at 184,284 size 326x28; TextOn '1'; TextOff '0'; TextList "007020_ASSIGNMENT_DIGITAL_OUTPUT"
      ProcessValue <- "WP231PR_DB_DR07_ASSIGN_DQ_3"
   Button "Schaltfläche_1" at 670,390 size 80x80; TextOn 'Texte'; TextOff 'Texte'; PictureOff "Q_Mark"
      on Press: SetBit("S1_SHOW_HELP")
   GraphicIOField "OBJECT_19" at 744,100 size 40x30; PictureList "Signal_grey_yellow"
      ProcessValue <- "WP231PR_DB_DR31_CURRENT_STATE_DQ_0"
   GraphicIOField "OBJECT_20" at 744,220 size 40x30; PictureList "Signal_grey_yellow"
      ProcessValue <- "WP231PR_DB_DR31_CURRENT_STATE_DQ_2"
   GraphicIOField "OBJECT_21" at 744,160 size 40x30; PictureList "Signal_grey_yellow"
      ProcessValue <- "WP231PR_DB_DR31_CURRENT_STATE_DQ_1"
   GraphicIOField "OBJECT_22" at 744,279 size 40x30; PictureList "Signal_grey_yellow"
      ProcessValue <- "WP231PR_DB_DR31_CURRENT_STATE_DQ_3"
   TextField "Textfeld_1" at 0,57 size 800x422; Text 'Um einen digitalen Ausgang direkt zu Steuern, muss ihm die Funktion "Test / Steuern Ausgang" zugewiesen werden! To test or force a digital output, the function of the corresponding output needs to be set to "Test / Force Output". Pour contrôler la sortie TOR il faut la choisir comme source'
      Visibility <- "S1_SHOW_HELP"
   Button "Schaltfläche_2" at 643,423 size 150x50; TextOn 'Texte'; TextOff 'OK'
      on Press: ResetBit("S1_SHOW_HELP")
      Visibility <- "S1_SHOW_HELP"

screen "1.5.0.2_Menu_communication_interfaces_2" 800x480, template "Template_1"
   TextField "OBJECT_82" at 0,0 size 709x34; Text '1.5.0 Kommunikation & Schnittstellen Seite 2 von 2 / 1.5.0 Communication & Interfaces 2 of 2 / 1.5.0 Communication et Interfaces 2/2 / Main Menu'
   Button "Password" at 33,174 size 350x90; TextOn 'Texte / text'; TextOff '1.5.8 Einstellungen Ethernet / 1.5.8 Ethernet Settings / 1.5.8 Paramétrage Ethernet / Diagnostics'
      on Press: ActivateScreen("0.0.0_Service_Ethernet", 0)
   Button "Expert calibration_1" at 33,73 size 350x90; TextOn 'Texte / text'; TextOff '1.5.7 Einstellungen Trace / 1.5.7 Trace Settings / 1.5.7 Paramétrage Trace / Enhanced Scale Setup'
      on Release: ActivateScreen("1.5.7_DR7_trace_settings", 0)
      on Press: SetTag("WP231PR_DB_s_CMD2_i_CMD_CODE", '2007'); SetBit("WP231PR_DB_s_CMD2_bo_CMD_TRIGGER")
   Button "Exit_to_Main_menue" at 45,390 size 80x80; TextOn 'Texte / text'; TextOff 'Texte / text'; PictureOff "Exit"
      on Press: ActivateScreen("1.0_Menu_setup", 0)
   Button "Exit_to_Main_menue_1" at 545,390 size 80x80; TextOn 'Texte / text'; TextOff 'Texte / text'; PictureOff "Left"
      on Press: ActivateScreen("1.5.0.1_Menu_communication_interfaces_1", 0)
   Button "Expert calibration_2" at 33,275 size 350x90; TextOn 'Texte / text'; TextOff '1.5.9 Einstellungen Simatic Schnittstelle 1.5.9 Simatic Interface Settings 1.5.9 Paramétrage SIMATIC Enhanced Scale Setup'
      on Release: ActivateScreen("1.5.9_DR14_S7_Interface_Parameter", 0)
      on Press: SetTag("WP231PR_DB_s_CMD2_i_CMD_CODE", '2014'); SetBit("WP231PR_DB_s_CMD2_bo_CMD_TRIGGER")
   Softkey "[!Invalid!]Softkey_F6" at -140,-147 size 0x0
      on KeyDown: ActivateScreen("1.0_Menu_setup", 0)

screen "0.0.0_Service_Quick_Start" 800x480, template "Template_1"
   Softkey "[!Invalid!]Softkey_F6" at -140,-147 size 0x0
      on KeyDown: SetTag("S1_CMD3.i_CMD_CODE", 2); SetTag("S1_CMD3.i_CMD_TRIGGER", 1); ActivateScreen("0.0.0_Menu_main", 0); function_efd93a16()
   Softkey "[!Invalid!]Softkey_F5" at -140,-147 size 0x0
      on KeyDown: SetTag("S1_CMD3.i_CMD_CODE", 1); SetTag("S1_CMD3.i_CMD_TRIGGER", 1); ActivateScreen("1.0_Menu_setup", 0)
   TextField "OBJECT_35" at 0,0 size 314x34; Text 'Quick Start - Warnung / Quick Start - Warning / Mise en service rapide / Calibration'
   Button "OBJECT_24" at 45,390 size 80x80; TextOn 'Texte / text'; TextOff 'Texte / text'; PictureOff "Exit"
      on Release: ActivateScreen("1.0_Menu_setup", 0)
      on Press: SetTag("WP231PR_DB_s_CMD2_i_CMD_CODE", 2); SetBit("WP231PR_DB_s_CMD2_bo_CMD_TRIGGER")
   TextField "OBJECT_1" at 24,89 size 127x33; Text 'Achtung! / Warning! / Attention / Calibration'
   TextField "OBJECT_2" at 20,119 size 773x120; Text 'Für "Quick Start" muss die Waage in den Service-Betrieb geschaltet werden. Sie haben Zugriff auf alle Waagenparameter! Der "Hilfe" Button der Touch-Tastatur beschreibt die Parameter. For "Quick Start" the scale needs to be in Serivce Mode. You will have full access to critical parameters! The "Help" button on the Touch-Keypad describes the single parameters. Mode service requis pour la mise en service rapide Calibration'
   Button "OBJECT_34" at 670,390 size 80x80; TextOn 'Texte / text'; TextOff 'Texte / text'; PictureOff "Right"
      on Release: ActivateScreen("1.2.1_Quick_Start_1", 0)
   Button "Service on_1" at 225,280 size 350x90; TextOn 'Texte / text'; TextOff 'Servicebetrieb einschalten Switch On "Service Mode" Mettre en mode service Acknowledge Empty Bin'
      on Press: SetTag("WP231PR_DB_s_CMD2_i_CMD_CODE", '1'); SetBit("WP231PR_DB_s_CMD2_bo_CMD_TRIGGER")
   Group "Group" at 700,5 size 95x30; Text 'Service'; PictureList "Signal_grey_yellow"
   GraphicIOField "OBJECT_19" at 765,5 size 30x30; PictureList "Signal_grey_yellow"
      ProcessValue <- "WP231PR_DB_s_IO_DATA_SCALE_STATUS_2_SERVICE_MODE"
   TextField "OBJECT_37" at 700,7 size 57x25; Text 'Service / Error occurred'

screen "1.2.7_Quick_Start_Automatic_Calibration" 800x480, template "Template_1"
   TextField "OBJECT_35" at 0,0 size 679x34; Text '1.2.7 Quick Start - Automatische Justage 5 von 5 / 1.2.7 Quick Start - Automatic Calibration 5 of 5 / 1.2.7 Mise en service rapide étalonnage auto 5/5 / Quick Setup'
   Button "Exit to Service" at 45,390 size 80x80; TextOn 'Texte / text'; TextOff 'Texte / text'; PictureOff "Exit"
      on Release: ActivateScreen("1.0_Menu_setup", 0); SetTag("WP231PR_DB_CMD_A", 2034)
      on Press: SetTag("WP231PR_DB_s_CMD2_i_CMD_CODE", '2'); SetBit("WP231PR_DB_s_CMD2_bo_CMD_TRIGGER")
   TextField "OBJECT_38" at 72,181 size 718x29; Text 'Für die automatische Justage muss die Waage jetzt leer sein ! / For automatic calibration the scale needs to be empty now! / La balance doit être vide pour l'étalonnage automatique / For Quick Setup the scale must be empty'
   Button "Confirm_scale_empty" at 110,236 size 580x70; TextOn 'Texte / text'; TextOff 'Automatische Justage durchführen / Start Automatic Calibration / Effectue l'étalonnage automatique / Acknowledge Empty Bin'
      on Release: SetTag("WP231PR_DB_s_CMD2_i_CMD_CODE", '2003'); SetBit("WP231PR_DB_s_CMD2_bo_CMD_TRIGGER")
      on Press: SetTag("WP231PR_DB_s_CMD1_i_CMD_CODE", '82'); SetBit("WP231PR_DB_s_CMD1_bo_CMD_TRIGGER")
   Button "Up_to Setup_5_Min_01" at 545,390 size 80x80; TextOn 'Texte / text'; TextOff 'Texte / text'; PictureOff "Left"
      on Release: ActivateScreen("1.2.6_Quick_Start_4", 0)
   Group "Group" at 700,5 size 95x30; Text 'Service'; PictureList "Signal_grey_yellow"
   IOField "OBJECT_301" at 0,74 size 800x86; FormatPattern ????????????????
      ProcessValue <- "WP231PR_DB_DR34_ASCII_DISPLAY"
   Button "Up_to Setup_5_Min_2" at 360,390 size 80x80; TextOn 'Texte / text'; TextOff 'Texte / text'; PictureOff "Home_3"
      on Release: ActivateScreen("0.0.0_Scale_View_1", 0); SetTag("WP231PR_DB_CMD_A", 2034)
      on Press: SetTag("WP231PR_DB_s_CMD2_i_CMD_CODE", '2'); SetBit("WP231PR_DB_s_CMD2_bo_CMD_TRIGGER")
   Softkey "[!Invalid!]Softkey_F6" at -140,-147 size 0x0
      on KeyDown: SetTag("S1_CMD3.i_CMD_CODE", 2); SetTag("S1_CMD3.i_CMD_TRIGGER", 1); ActivateScreen("1.0_Menu_setup", 0)
   Softkey "[!Invalid!]Softkey_F4" at -140,-147 size 0x0
      on KeyDown: ActivateScreen("1.2.6_Quick_Start_4", 0)
   GraphicIOField "OBJECT_19" at 765,5 size 30x30; PictureList "Signal_grey_yellow"
      ProcessValue <- "WP231PR_DB_s_IO_DATA_SCALE_STATUS_2_SIMULATION_MODE"
   TextField "OBJECT_37" at 700,7 size 57x25; Text 'Service / Error occurred'

screen "1.2.2_Quick_Start_2" 800x480, template "Template_1"
   TextField "OBJECT_33" at 0,0 size 440x34; Text '1.2.2 Quick Start 2 von 5 / 1.2.2 Quick Start 2 of 5 / 1.2.2 Mise en service rapide 2/5 / Setup 1/3'
   Button "Exit to Service" at 45,390 size 80x80; TextOn 'Texte / text'; TextOff 'Texte / text'; PictureOff "Exit"
      on Release: ActivateScreen("1.0_Menu_setup", 0)
      on Press: SetTag("WP231PR_DB_s_CMD2_i_CMD_CODE", '2'); SetBit("WP231PR_DB_s_CMD2_bo_CMD_TRIGGER")
   Group "Group" at 700,5 size 95x30; Text 'Service'; PictureList "Signal_grey_yellow"
   TextField "OBJECT_306" at 234,90 size 179x29; Text 'Waagenname / Scale Name / Nom de la balance / Scale name'
   IOField "OBJECT_307" at 420,84 size 172x40; HelpText 'Name der Waage (Produkt, Anlagenteil o.Ä.) / Nom de la balance'; FormatPattern ????????????
      ProcessValue <- "WP231PR_DB_DR03_SCALE_NAME"
   TextField "OBJECT_7" at 258,141 size 151x29; Text 'Gewichtseinheit / Weight unit / Unité poids / Weight Unit'
   IOField "OBJECT_28" at 420,134 size 172x40; HelpText 'Gewichtseinheit (z.B. g, kg oder t) / Unité poids (par ex. g, kg ou t)'; FormatPattern ????
      ProcessValue <- "WP231PR_DB_DR03_WEIGHT_UNIT"
   TextField "OBJECT_9" at 129,285 size 283x29; Text 'Minimaler Wägebereich (in d) / Minimum weight (in d) / Poids min (en d) / Weight Unit'
   TextField "OBJECT_10" at 159,330 size 254x29; Text 'Maximaler Wägebereich / Maximum weight / Plage maximale de pesage / Weight Unit'
   TextField "OBJECT_11" at 252,237 size 159x29; Text 'Ziffernschritt (d) / Resolution / Résolution (d) / Weight Unit'
   IOField "OBJECT_29" at 420,279 size 172x40; HelpText 'Bei geeichten Waagen mind. 20 x Ziffernschritt d. Bei nicht eichpflichtigen Waagen kann der minimale Wägebereich mit 0 definiert werden. / 20 x d pour usage certifié, sinon pas de limitation (0 par exemple)'; FormatPattern 999
      ProcessValue <- "WP231PR_DB_DR03_MIN_WEIGHT_D"
   IOField "OBJECT_12" at 420,325 size 173x40; HelpText 'Maximales Gewicht auf der Waage. Bei geeichten Waagen bitte entsprechende Einschränkungen beachten! / Poids max. sur la balance'; FormatPattern 9999999.9999
      ProcessValue <- "WP231PR_DB_DR03_MAX_WEIGHT"
   IOField "OBJECT_13" at 420,230 size 172x40; HelpText 'Ziffernschritt der Waage. Ist die Gewichts einheit "kg" bedeutet ein Ziffernschritt von 0,1 dass die Waage in 0,1kg Schritten auflöst. / Résolution de la balance. Avec un unité de poids de 1kg, la résolution de 0,1 signifie 0,1kg'; FormatPattern 9999.9999
      ProcessValue <- "WP231PR_DB_DR03_RESOLUTION_D"
   IOField "I/O field_2" at 596,325 size 60x40; FormatPattern ????
      ProcessValue <- "WP231PR_DB_DR03_WEIGHT_UNIT"
   TextField "Textfeld_1" at 609,283 size 18x29; Text 'x'
   Group "Group_1" at 607,242 size 62x59
   Button "Down to Setup_5_Min_03" at 690,390 size 80x80; TextOn 'Texte / text'; TextOff 'Texte / text'; PictureOff "Right"
      on Release: ActivateScreen("1.2.3_Quick_Start_3", 0)
   Button "Up_to Setup_5_Min_01" at 545,390 size 80x80; TextOn 'Texte / text'; TextOff 'Texte / text'; PictureOff "Left"
      on Release: ActivateScreen("1.2.1_Quick_Start_1", 0)
   TextField "OBJECT_6" at 8,188 size 403x29; Text 'Brutto-Kennung ("B" oder "G") / Indicator for Gross ("B" or "G") / Abréviation pour le poids brut ("B" ou "G") / Weight Unit'
   SymbolicIOField "Symbolic I/O field_1" at 421,187 size 172x31; TextOn '1'; TextOff '0'; TextList "003030_LETTER_FOR_GROSS_WEIGHT"
      ProcessValue <- "WP231PR_DB_DR03_LETTER_GROSS_WEIGHT_2"
   Button "Down to Setup_5_Min_1" at 360,390 size 80x80; TextOn 'Texte / text'; TextOff 'Texte / text'; PictureOff "Save"
      on Press: SetTag("WP231PR_DB_s_CMD2_i_CMD_CODE", '4003'); SetBit("WP231PR_DB_s_CMD2_bo_CMD_TRIGGER")
   Softkey "[!Invalid!]Softkey_F6" at -140,-147 size 0x0
      on KeyDown: ActivateScreen("1.0_Menu_setup", 0)
   Softkey "[!Invalid!]Softkey_F5" at -140,-147 size 0x0
      on KeyDown: SetTag("S1_CMD2.i_CMD_CODE", 2010); SetTag("S1_CMD2.i_CMD_TRIGGER", 1); SetTag("S1_CMD3.i_CMD_CODE", 2003); SetTag("S1_CMD3.i_CMD_TRIGGER", 1); ActivateScreen("1.2.6_Quick_Start_4", 0)
   GraphicIOField "OBJECT_19" at 765,5 size 30x30; PictureList "Signal_grey_yellow"
      ProcessValue <- "WP231PR_DB_s_IO_DATA_SCALE_STATUS_2_SIMULATION_MODE"
   TextField "OBJECT_37" at 700,7 size 57x25; Text 'Service / Error occurred'

screen "1.2.4_Quick_Start_Manual_Calibration_1" 800x480, template "Template_1"
   TextField "OBJECT_33" at 0,0 size 630x34; Text '1.2.4 Quick Start - Justagegewichte 4 von 5 / 1.2.4 Quick Start - Calibration Weights 4 of 5 / 1.2.4 Mise en service rapide poids étalon 4/5 / Setup 1/3'
   TextField "OBJECT_306" at 157,135 size 206x32; Text 'Justagegewicht 0 / Calibration weight 0 / Poids étalon 0 / Scale name'
   Button "OBJECT_34" at 670,390 size 80x80; TextOn 'Texte / text'; TextOff 'Texte / text'; PictureOff "Right"
      on Release: ActivateScreen("1.2.5_Quick_Start_Manual_Calibration_2", 0); SetTag("WP231PR_DB_CMD_A", 2034)
      on Press: SetTag("WP231PR_DB_CMD_B", 2031)
   IOField "OBJECT_307" at 373,126 size 300x50; HelpText 'Falls die Waage zum Zeitpunkt der Justage nicht leer ist, kann das bekannte Gewicht in der Waage als "Justagegewicht 0" vorgegeben werden. / If the scale is not empty before adjusting, the known material weight in the scale can be defined as "Calibration weight 0". / Si pour l'étalonnage la balance n'est pas vide, il est possible d'utiliser le poids actuel comme poids étalon'; FormatPattern 999999.999
      ProcessValue <- "WP231PR_DB_DR03_CALIB_WEIGHT_0"
   TextField "OBJECT_7" at 158,192 size 206x32; Text 'Justagegewicht 1 / Calibration weight 1 / Poids étalon 1 / Weight Unit'
   IOField "OBJECT_28" at 373,182 size 300x50; HelpText 'Das "Justagegewicht 1" muss mindestens 5% der Nennlast der Waage entsprechen! / Le poids étalon doit être supérieur à 5% de la charge max des pesons'; FormatPattern 999999.999
      ProcessValue <- "WP231PR_DB_DR03_CALIB_WEIGHT_1"
   Button "OBJECT_24" at 45,390 size 80x80; TextOn 'Texte / text'; TextOff 'Texte / text'; PictureOff "Exit"
      on Release: ActivateScreen("1.0_Menu_setup", 0)
      on Press: SetTag("WP231PR_DB_s_CMD2_i_CMD_CODE", '2'); SetBit("WP231PR_DB_s_CMD2_bo_CMD_TRIGGER")
   TextField "OBJECT_6" at 42,248 size 320x32; Text 'Justagegewicht 2 (optional) / Calibration weight 2 (optional) / Poids étalon 2 (option) / Weight Unit'
   IOField "OBJECT_8" at 372,240 size 302x50; HelpText 'Mit "Justagegewicht 2" kann ein dritter Justagepunkt gesetzt werden. Es ist nicht zwingend erforderlich diesen zu setzen! Falls genutzt, muss der Abstand zwischen "Justagegewicht 1" und "Justagegewicht 2" mind. 5% der Nennlast der Waage entsprechen. Le poids étalon 2 permet d'avoir un troisième points d'étalonnage'; FormatPattern 999999.999
      ProcessValue <- "WP231PR_DB_DR03_CALIB_WEIGHT_2"
   IOField "I/O field_2" at 676,131 size 60x40; FormatPattern ????
      ProcessValue <- "WP231PR_DB_DR03_WEIGHT_UNIT"
   IOField "I/O field_1" at 676,189 size 60x40; FormatPattern ????
      ProcessValue <- "WP231PR_DB_DR03_WEIGHT_UNIT"
   IOField "I/O field_3" at 677,244 size 60x40; FormatPattern ????
      ProcessValue <- "WP231PR_DB_DR03_WEIGHT_UNIT"
   Group "Group" at 700,5 size 95x30; Text 'Service'; PictureList "Signal_grey_yellow"
   Button "Up_to Setup_5_Min_01" at 545,390 size 80x80; TextOn 'Texte / text'; TextOff 'Texte / text'; PictureOff "Left"
      on Release: ActivateScreen("1.2.3_Quick_Start_3", 0)
   Button "Schaltfläche_1" at 213,390 size 80x80; TextOn 'Texte'; TextOff 'Texte'; PictureOff "Q_Mark"
      on Press: SetBit("S1_SHOW_HELP")
   Button "OBJECT_1" at 360,390 size 80x80; TextOn 'Texte / text'; TextOff 'Texte / text'; PictureOff "Save"
      on Press: SetTag("WP231PR_DB_s_CMD2_i_CMD_CODE", '4003'); SetBit("WP231PR_DB_s_CMD2_bo_CMD_TRIGGER")
   Softkey "[!Invalid!]Softkey_F6" at -140,-147 size 0x0
      on KeyDown: ActivateScreen("Menu_weighing_expert", 0)
   Softkey "[!Invalid!]Softkey_F5" at -140,-147 size 0x0
      on KeyDown: SetTag("S1_CMD2.i_CMD_CODE", 4003); SetTag("S1_CMD2.i_CMD_TRIGGER", 1); ActivateScreen("Calibration", 0); SetTag("S1_CMD2.i_CMD_CODE", 4003); SetTag("S1_CMD2.i_CMD_TRIGGER", 1); ActivateScreen("Calibration", 0)
   GraphicIOField "OBJECT_19" at 765,5 size 30x30; PictureList "Signal_grey_yellow"
      ProcessValue <- "WP231PR_DB_s_IO_DATA_SCALE_STATUS_2_SIMULATION_MODE"
   TextField "OBJECT_37" at 700,7 size 57x25; Text 'Service / Error occurred'
   GraphicView "Grafikanzeige_1" at 4,7 size 793x470; Picture "char_curve"
      Visibility <- "S1_SHOW_HELP"
   Button "Schaltfläche_2" at 19,420 size 150x50; TextOn 'Texte'; TextOff 'OK'
      on Press: ResetBit("S1_SHOW_HELP")
      Visibility <- "S1_SHOW_HELP"

screen "1.2.5_Quick_Start_Manual_Calibration_2" 800x480, template "Template_1"
   TextField "OBJECT_35" at 0,0 size 691x34; Text '1.2.5 Quick Start - Justage mit Gewichten 5 von 5 / 1.2.5 Quick Start - Calibration with Weights / 1.2.5 Mise en service rapide poids étalon 5/5 / Calibration'
   IOField "OBJECT_301" at 0,41 size 800x90; FormatPattern ????????????????
      ProcessValue <- "WP231PR_DB_DR34_ASCII_DISPLAY"
   Group "Group" at 700,5 size 95x30; Text 'Service'; PictureList "Signal_grey_yellow"
   Button "Up_to Setup_5_Min_01" at 545,390 size 80x80; TextOn 'Texte / text'; TextOff 'Texte / text'; PictureOff "Left"
      on Release: ActivateScreen("1.2.4_Quick_Start_Manual_Calibration_1", 0); SetTag("WP231PR_DB_CMD_A", 2034)
      on Press: SetTag("WP231PR_DB_s_CMD2_i_CMD_CODE", '2003'); SetBit("WP231PR_DB_s_CMD2_bo_CMD_TRIGGER"); SetTag("WP231PR_DB_CMD_B", 0)
   Button "Exit to Service" at 45,390 size 80x80; TextOn 'Texte / text'; TextOff 'Texte / text'; PictureOff "Exit"
      on Release: ActivateScreen("1.0_Menu_setup", 0); SetTag("WP231PR_DB_CMD_A", 2034); SetTag("WP231PR_DB_s_CMD1_i_CMD_CODE", '2'); SetBit("WP231PR_DB_s_CMD1_bo_CMD_TRIGGER")
      on Press: SetTag("WP231PR_DB_s_CMD2_i_CMD_CODE", '2'); SetBit("WP231PR_DB_s_CMD2_bo_CMD_TRIGGER"); SetTag("WP231PR_DB_CMD_B", 0)
   Button "OBJECT_28" at 110,135 size 580x70; TextOn 'Texte / text'; TextOff 'Justagegewicht 0 setzen / Set Calibration Weight 0 / Placez le poids étalon 0 / Acknowledge Empty Bin'
      on Press: SetTag("WP231PR_DB_s_CMD2_i_CMD_CODE", '60'); SetBit("WP231PR_DB_s_CMD2_bo_CMD_TRIGGER")
   Button "OBJECT_31" at 110,207 size 580x70; TextOn 'Texte / text'; TextOff 'Justagegewicht 1 setzen / Set Calibration Weight 1 / Placez le poids étalon 1 / Put & Acknowledge Calibration Weight'
      on Press: SetTag("WP231PR_DB_s_CMD2_i_CMD_CODE", '61'); SetBit("WP231PR_DB_s_CMD2_bo_CMD_TRIGGER")
   Button "Up_to Setup_5_Min_2" at 360,390 size 80x80; TextOn 'Texte / text'; TextOff 'Texte / text'; PictureOff "Home_3"
      on Release: ActivateScreen("0.0.0_Scale_View_1", 0); SetTag("WP231PR_DB_CMD_A", 2034)
      on Press: SetTag("WP231PR_DB_s_CMD2_i_CMD_CODE", '2'); SetBit("WP231PR_DB_s_CMD2_bo_CMD_TRIGGER"); SetTag("WP231PR_DB_CMD_B", 0)
   Button "OBJECT_3" at 110,279 size 580x70; TextOn 'Texte / text'; TextOff 'Justagegewicht 2 setzen (optional) / Set Calibration Weight 2 (optional) / Placez le poids étalon 2 (option) / Put & Acknowledge Calibration Weight'
      on Press: SetTag("WP231PR_DB_s_CMD2_i_CMD_CODE", '62'); SetBit("WP231PR_DB_s_CMD2_bo_CMD_TRIGGER")
   Softkey "[!Invalid!]Softkey_F6" at -140,-147 size 0x0
      on KeyDown: ActivateScreen("Menu_weighing_expert", 0)
   Softkey "[!Invalid!]Softkey_F5" at -140,-147 size 0x0
      on KeyDown: ActivateScreen("DR3_Calibration weights", 0)
   GraphicIOField "OBJECT_19" at 765,5 size 30x30; PictureList "Signal_grey_yellow"
      ProcessValue <- "WP231PR_DB_s_IO_DATA_SCALE_STATUS_2_SIMULATION_MODE"
   TextField "OBJECT_37" at 700,7 size 57x25; Text 'Service / Error occurred'
   TextField "OBJECT_4" at 227,352 size 207x32; Text 'Aktuelle Digits ADC: / Current ADC digits: / Valeur CAN / Error occurred'
   IOField "I/O field_5" at 442,352 size 136x32; FormatPattern 9999999999
      ProcessValue <- "WP231PR_DB_DR31_DIGITS_FILTERED"

screen "2.3.0_Load_Trend" 800x480, template "Template_1"
   TrendView "Kurvenanzeige_1" at 0,48 size 710x426
      ValueAxis1End <- "WP231PR_DB_DR03_MAX_WEIGHT"
      ValueAxis1Begin <- "S1_LOADCURVE_MIN"
   IOField "EA-Feld_1" at 48,7 size 110x35; FormatPattern 9999999999
      ProcessValue <- "S1_LOADCURVE_MIN"
   IOField "EA-Feld_2" at 273,6 size 103x35; FormatPattern 999999999
      ProcessValue <- "WP231PR_DB_DR03_MAX_WEIGHT"
   Button "Exit_to_Main_menue" at 715,390 size 80x80; TextOn 'Texte / text'; TextOff 'Texte / text'; PictureOff "Exit"
      on Release: ActivateScreen("2.0_Menu_diagnostic", 0)
      on Press: SetTag("WP231PR_DB_CMD_B", 0)
   IOField "OBJECT_301" at 538,3 size 259x40; FormatPattern s999999999.999
      ProcessValue <- "WP231PR_DB_DR30_GROSS_PROCESS"
   TextField "Textfeld_1" at 227,11 size 39x25; Text 'Max.'
   TextField "Textfeld_2" at 5,11 size 35x25; Text 'Min. / Min'
   IOField "EA-Feld_3" at 161,11 size 66x25; FormatPattern ????
      ProcessValue <- "WP231PR_DB_DR03_WEIGHT_UNIT"
   IOField "EA-Feld_4" at 378,11 size 66x25; FormatPattern ????
      ProcessValue <- "WP231PR_DB_DR03_WEIGHT_UNIT"
   TextField "Textfeld_3" at 486,11 size 50x25; Text 'Brutto / Gross / Brut'

screen "0.0.0_Service_Adv_Scale_Para" 800x480, template "Template_1"
   Softkey "[!Invalid!]Softkey_F6" at -140,-147 size 0x0
      on KeyDown: SetTag("S1_CMD3.i_CMD_CODE", 2); SetTag("S1_CMD3.i_CMD_TRIGGER", 1); ActivateScreen("0.0.0_Menu_main", 0); function_efd93a16()
   Softkey "[!Invalid!]Softkey_F5" at -140,-147 size 0x0
      on KeyDown: SetTag("S1_CMD3.i_CMD_CODE", 1); SetTag("S1_CMD3.i_CMD_TRIGGER", 1); ActivateScreen("1.0_Menu_setup", 0)
   TextField "OBJECT_35" at 0,0 size 563x34; Text 'Erweiterte Waagenparameter - Warnung / Advanced Scale Settings - Warning / Paramètres balances / Calibration'
   Button "OBJECT_24" at 45,390 size 80x80; TextOn 'Texte / text'; TextOff 'Texte / text'; PictureOff "Exit"
      on Release: ActivateScreen("1.0_Menu_setup", 0)
      on Press: SetTag("WP231PR_DB_s_CMD2_i_CMD_CODE", 2); SetBit("WP231PR_DB_s_CMD2_bo_CMD_TRIGGER")
   TextField "OBJECT_1" at 24,89 size 127x33; Text 'Achtung! / Warning! / Attention / Calibration'
   TextField "OBJECT_2" at 24,122 size 773x122; Text 'Für weitere Schritte muss die Waage in den Service-Betrieb geschaltet werden. Sie haben Zugriff auf alle Waagenparameter! Der "Hilfe" Button der Touch-Tastatur beschreibt die Parameter. For further steps the scale needs to be in Serivce Mode. You will have full access to critical parameters! The "Help" button on the Touch-Keypad describes the single parameters. Mode service requis pour les étapes suivantes Calibration'
   Button "OBJECT_34" at 670,390 size 80x80; TextOn 'Texte / text'; TextOff 'Texte / text'; PictureOff "Right"
      on Release: ActivateScreen("1.4.1_DR3_Advanced_Scale_Parameters_1", 0)
      on Press: SetTag("WP231PR_DB_s_CMD2_i_CMD_CODE", '2003'); SetBit("WP231PR_DB_s_CMD2_bo_CMD_TRIGGER")
   Button "Service on_1" at 225,280 size 350x90; TextOn 'Texte / text'; TextOff 'Servicebetrieb einschalten Switch On "Service Mode" Mettre en mode service Acknowledge Empty Bin'
      on Press: SetTag("WP231PR_DB_s_CMD2_i_CMD_CODE", '1'); SetBit("WP231PR_DB_s_CMD2_bo_CMD_TRIGGER")
   Group "Group" at 700,5 size 95x30; Text 'Service'; PictureList "Signal_grey_yellow"
   GraphicIOField "OBJECT_19" at 765,5 size 30x30; PictureList "Signal_grey_yellow"
      ProcessValue <- "WP231PR_DB_s_IO_DATA_SCALE_STATUS_2_SERVICE_MODE"
   TextField "OBJECT_37" at 700,7 size 57x25; Text 'Service / Error occurred'

screen "0.0.0_Service_Recovery" 800x480, template "Template_1"
   Softkey "[!Invalid!]Softkey_F6" at -140,-147 size 0x0
      on KeyDown: SetTag("S1_CMD3.i_CMD_CODE", 2); SetTag("S1_CMD3.i_CMD_TRIGGER", 1); ActivateScreen("0.0.0_Menu_main", 0); function_efd93a16()
   Softkey "[!Invalid!]Softkey_F5" at -140,-147 size 0x0
      on KeyDown: SetTag("S1_CMD3.i_CMD_CODE", 1); SetTag("S1_CMD3.i_CMD_TRIGGER", 1); ActivateScreen("1.0_Menu_setup", 0)
   TextField "OBJECT_35" at 0,0 size 635x34; Text 'Wiederherstellung - Warnung / Recovery - Warning / Recharger avec les paramètres de sauvegarde / Calibration'
   Button "OBJECT_24" at 45,390 size 80x80; TextOn 'Texte / text'; TextOff 'Texte / text'; PictureOff "Exit"
      on Release: ActivateScreen("1.0_Menu_setup", 0)
      on Press: SetTag("WP231PR_DB_s_CMD2_i_CMD_CODE", 2); SetBit("WP231PR_DB_s_CMD2_bo_CMD_TRIGGER")
   TextField "OBJECT_1" at 24,89 size 127x33; Text 'Achtung! / Warning! / Attention / Calibration'
   TextField "OBJECT_2" at 18,126 size 782x108; Text 'Für die Wiederherstellungs-Funktionen muss die Waage in den Service- Betrieb geschaltet werden. Sie haben Zugriff auf alle Waagenparameter. Die aktuellen Waagenparameter können überschrieben werden! Der "Hilfe" Button der Touch-Tastatur beschreibt die einzelnen Optionen. For "Recovery" the scale needs to be in Service Mode. You will have full access to all critical parameters. Important scale settings might be overwritten! The "Help" button on the Touch-Keypad describes the different options. Mode service requis pour la réécriture des paramètres Calibration'
   Button "OBJECT_34" at 670,390 size 80x80; TextOn 'Texte / text'; TextOff 'Texte / text'; PictureOff "Right"
      on Press: ActivateScreen("1.6.1_Recovery_point", 0)
   Button "Service on_1" at 225,280 size 350x90; TextOn 'Texte / text'; TextOff 'Servicebetrieb einschalten Switch On "Service Mode" Mettre en mode service Acknowledge Empty Bin'
      on Press: SetTag("WP231PR_DB_s_CMD2_i_CMD_CODE", '1'); SetBit("WP231PR_DB_s_CMD2_bo_CMD_TRIGGER")
   Group "Group" at 700,5 size 95x30; Text 'Service'; PictureList "Signal_grey_yellow"
   GraphicIOField "OBJECT_19" at 765,5 size 30x30; PictureList "Signal_grey_yellow"
      ProcessValue <- "WP231PR_DB_s_IO_DATA_SCALE_STATUS_2_SERVICE_MODE"
   TextField "OBJECT_37" at 700,7 size 57x25; Text 'Service / Error occurred'

screen "0.0.0_Service_Ethernet" 800x480, template "Template_1"
   Softkey "[!Invalid!]Softkey_F6" at -140,-147 size 0x0
      on KeyDown: SetTag("S1_CMD3.i_CMD_CODE", 2); SetTag("S1_CMD3.i_CMD_TRIGGER", 1); ActivateScreen("0.0.0_Menu_main", 0); function_efd93a16()
   Softkey "[!Invalid!]Softkey_F5" at -140,-147 size 0x0
      on KeyDown: SetTag("S1_CMD3.i_CMD_CODE", 1); SetTag("S1_CMD3.i_CMD_TRIGGER", 1); ActivateScreen("1.0_Menu_setup", 0)
   TextField "OBJECT_35" at 0,0 size 563x34; Text 'Erweiterte Waagenparameter - Warnung / Advanced Scale Settings - Warning / Paramètres balances / Calibration'
   Button "OBJECT_24" at 45,390 size 80x80; TextOn 'Texte / text'; TextOff 'Texte / text'; PictureOff "Exit"
      on Release: ActivateScreen("1.5.0.2_Menu_communication_interfaces_2", 0)
      on Press: SetTag("WP231PR_DB_s_CMD2_i_CMD_CODE", 2); SetBit("WP231PR_DB_s_CMD2_bo_CMD_TRIGGER")
   TextField "OBJECT_1" at 24,89 size 127x33; Text 'Achtung! / Warning! / Attention / Calibration'
   TextField "OBJECT_2" at 14,122 size 771x120; Text 'Für weitere Schritte muss die Waage in den Service-Betrieb geschaltet werden. Sie haben Zugriff auf alle Waagenparameter! Der "Hilfe" Button der Touch-Tastatur beschreibt die Parameter. For further steps the scale needs to be in Serivce Mode. You will have full access to critical parameters! The "Help" button on the Touch-Keypad describes the single parameters. Mode service requis pour les étapes suivantes Calibration'
   Button "OBJECT_34" at 670,390 size 80x80; TextOn 'Texte / text'; TextOff 'Texte / text'; PictureOff "Right"
      on Release: ActivateScreen("1.5.8_DR12_Ethernet_parameters", 0)
      on Press: SetTag("WP231PR_DB_s_CMD2_i_CMD_CODE", '2012'); SetBit("WP231PR_DB_s_CMD2_bo_CMD_TRIGGER")
   Button "Service on_1" at 225,280 size 350x90; TextOn 'Texte / text'; TextOff 'Servicebetrieb einschalten Switch On "Service Mode" Mettre en mode service Acknowledge Empty Bin'
      on Press: SetTag("WP231PR_DB_s_CMD2_i_CMD_CODE", '1'); SetBit("WP231PR_DB_s_CMD2_bo_CMD_TRIGGER")
   Group "Group" at 700,5 size 95x30; Text 'Service'; PictureList "Signal_grey_yellow"
   GraphicIOField "OBJECT_19" at 765,5 size 30x30; PictureList "Signal_grey_yellow"
      ProcessValue <- "WP231PR_DB_s_IO_DATA_SCALE_STATUS_2_SERVICE_MODE"
   TextField "OBJECT_37" at 700,7 size 57x25; Text 'Service / Error occurred'
*)

(* ===== HMI "HMI_RT_1" =====
system functions are stored by id; their names below are inferred from use
connection "HMI_Connection_1": ETHERNET, SMART_S7_1200_OMS

